LIN {X 0,Y 394.294,Z 695.223,A -85,B 0,C 180,E1 18299.135,E2 18299.135} C_VEL
LIN {X 0,Y 391.517,Z 710.275,A -85,B 0,C 180,E1 18296.546,E2 18296.546} C_VEL
LIN {X 0,Y 389.156,Z 723.905,A -85,B 0,C 180,E1 18293.789,E2 18293.789} C_VEL
LIN {X 0,Y 387.17,Z 736.546,A -85,B 0,C 180,E1 18290.72,E2 18290.72} C_VEL
LIN {X 0,Y 385.749,Z 746.976,A -85,B 0,C 180,E1 18287.654,E2 18287.654} C_VEL
LIN {X 0,Y 384.84,Z 755.495,A -85,B 0,C 180,E1 18284.597,E2 18284.597} C_VEL
LIN {X 0,Y 384.288,Z 762.773,A -85,B 0,C 180,E1 18281.253,E2 18281.253} C_VEL
LIN {X 0,Y 384.081,Z 767.655,A -85,B 0,C 180,E1 18278.232,E2 18278.232} C_VEL
LIN {X 0,Y 384.027,Z 771.125,A -85,B 0,C 180,E1 18275.078,E2 18275.078} C_VEL
LIN {X 0,Y 384.034,Z 772.853,A -85,B 0,C 180,E1 18272.089,E2 18272.089} C_VEL
LIN {X 0,Y 384.041,Z 773.096,A -85,B 0,C 180,E1 18268.956,E2 18268.956} C_VEL
LIN {X 0,Y 384.03,Z 771.796,A -85,B 0,C 180,E1 18265.969,E2 18265.969} C_VEL
LIN {X 0,Y 384.061,Z 768.821,A -85,B 0,C 180,E1 18262.821,E2 18262.821} C_VEL
LIN {X 0,Y 384.195,Z 764.382,A -85,B 0,C 180,E1 18259.807,E2 18259.807} C_VEL
LIN {X 0,Y 384.596,Z 757.969,A -85,B 0,C 180,E1 18256.621,E2 18256.621} C_VEL
LIN {X 0,Y 385.379,Z 749.606,A -85,B 0,C 180,E1 18253.417,E2 18253.417} C_VEL
LIN {X 0,Y 386.587,Z 739.686,A -85,B 0,C 180,E1 18250.352,E2 18250.352} C_VEL
LIN {X 0,Y 388.331,Z 727.636,A -85,B 0,C 180,E1 18247.281,E2 18247.281} C_VEL
LIN {X 0,Y 390.438,Z 714.67,A -85,B 0,C 180,E1 18244.518,E2 18244.518} C_VEL
LIN {X 0,Y 393.123,Z 699.469,A -85,B 0,C 180,E1 18241.766,E2 18241.766} C_VEL
LIN {X 0,Y 396.114,Z 683.012,A -85,B 0,C 180,E1 18239.26,E2 18239.26} C_VEL
LIN {X 0,Y 399.307,Z 665.741,A -85,B 0,C 180,E1 18237.017,E2 18237.017} C_VEL
LIN {X 0,Y 402.758,Z 646.554,A -85,B 0,C 180,E1 18234.921,E2 18234.921} C_VEL
LIN {X 0,Y 406.358,Z 625.751,A -85,B 0,C 180,E1 18233.015,E2 18233.015} C_VEL
LIN {X 0,Y 410.133,Z 603.324,A -85,B 0,C 180,E1 18231.294,E2 18231.294} C_VEL
LIN {X 0,Y 413.644,Z 580.978,A -85,B 0,C 180,E1 18229.895,E2 18229.895} C_VEL
LIN {X 0,Y 417.206,Z 557.129,A -85,B 0,C 180,E1 18228.681,E2 18228.681} C_VEL
LIN {X 0,Y 420.545,Z 532.633,A -85,B 0,C 180,E1 18227.713,E2 18227.713} C_VEL
LIN {X 0,Y 423.355,Z 506.29,A -85,B 0,C 180,E1 18226.922,E2 18226.922} C_VEL
LIN {X 0,Y 425.187,Z 485.655,A -85,B 0,C 180,E1 18226.474,E2 18226.474} C_VEL
LIN {X 0,Y 427.43,Z 463.252,A -85,B 0,C 180,E1 18226.233,E2 18226.233} C_VEL
LIN {X 0,Y 430.001,Z 440.333,A -85,B 0,C 180,E1 18226.045,E2 18226.045} C_VEL
LIN {X 0,Y 437.672,Z 418.91,A -85,B 0,C 180,E1 18225.373,E2 18225.373} C_VEL
LIN {X 0,Y 445.295,Z 397.451,A -85,B 0,C 180,E1 18224.711,E2 18224.711} C_VEL
LIN {X 0,Y 455.695,Z 372.925,A -85,B 0,C 180,E1 18224.152,E2 18224.152} C_VEL
LIN {X 0,Y 470.521,Z 341.939,A -85,B 0,C 180,E1 18223.651,E2 18223.651} C_VEL
LIN {X 0,Y 460.391,Z 331.053,A -85,B 0,C 180,E1 18221.815,E2 18221.815} C_VEL
LIN {X 0,Y 451.953,Z 318.726,A -85,B 0,C 180,E1 18219.908,E2 18219.908} C_VEL
LIN {X 0,Y 445.362,Z 304.779,A -85,B 0,C 180,E1 18217.962,E2 18217.962} C_VEL
LIN {X 0,Y 440.291,Z 291.135,A -85,B 0,C 180,E1 18216.107,E2 18216.107} C_VEL
LIN {X 0,Y 426.278,Z 299.916,A -85,B 0,C 180,E1 18214.584,E2 18214.584} C_VEL
LIN {X 0,Y 421.514,Z 303.016,A -85,B 0,C 180,E1 18214.042,E2 18214.042} C_VEL
LIN {X 0,Y 419.973,Z 303.956,A -85,B 0,C 180,E1 18213.855,E2 18213.855} C_VEL
LIN {X 0,Y 415.952,Z 306.923,A -85,B 0,C 180,E1 18213.399,E2 18213.399} C_VEL
LIN {X 0,Y 413.79,Z 308.018,A -85,B 0,C 180,E1 18213.099,E2 18213.099} C_VEL
LIN {X 0,Y 410.423,Z 310.916,A -85,B 0,C 180,E1 18212.74,E2 18212.74} C_VEL
LIN {X 0,Y 407.643,Z 312.19,A -85,B 0,C 180,E1 18212.324,E2 18212.324} C_VEL
LIN {X 0,Y 407.314,Z 312.632,A -85,B 0,C 180,E1 18212.228,E2 18212.228} C_VEL
LIN {X 0,Y 405.552,Z 347.302,A -85,B 0,C 180,E1 18208.976,E2 18208.976} C_VEL
LIN {X 0,Y 402.812,Z 358.585,A -85,B 0,C 180,E1 18208.28,E2 18208.28} C_VEL
LIN {X 0,Y 397.59,Z 457.682,A -85,B 0,C 180,E1 18205.679,E2 18205.679} C_VEL
LIN {X 0,Y 396.033,Z 507.95,A -85,B 0,C 180,E1 18204.434,E2 18204.434} C_VEL
LIN {X 0,Y 395.904,Z 528.625,A -85,B 0,C 180,E1 18203.798,E2 18203.798} C_VEL
LIN {X 0,Y 395.515,Z 545.902,A -85,B 0,C 180,E1 18202.998,E2 18202.998} C_VEL
LIN {X 0,Y 394.84,Z 562.776,A -85,B 0,C 180,E1 18201.932,E2 18201.932} C_VEL
LIN {X 0,Y 393.999,Z 577.422,A -85,B 0,C 180,E1 18200.732,E2 18200.732} C_VEL
LIN {X 0,Y 392.965,Z 591.658,A -85,B 0,C 180,E1 18199.269,E2 18199.269} C_VEL
LIN {X 0,Y 391.833,Z 604.688,A -85,B 0,C 180,E1 18197.6,E2 18197.6} C_VEL
LIN {X 0,Y 390.654,Z 616.279,A -85,B 0,C 180,E1 18195.741,E2 18195.741} C_VEL
LIN {X 0,Y 389.573,Z 625.958,A -85,B 0,C 180,E1 18193.809,E2 18193.809} C_VEL
LIN {X 0,Y 388.598,Z 634.231,A -85,B 0,C 180,E1 18191.728,E2 18191.728} C_VEL
LIN {X 0,Y 387.758,Z 641.05,A -85,B 0,C 180,E1 18189.498,E2 18189.498} C_VEL
LIN {X 0,Y 387.046,Z 646.284,A -85,B 0,C 180,E1 18187.122,E2 18187.122} C_VEL
LIN {X 0,Y 386.544,Z 649.693,A -85,B 0,C 180,E1 18184.747,E2 18184.747} C_VEL
LIN {X 0,Y 386.218,Z 651.422,A -85,B 0,C 180,E1 18182.373,E2 18182.373} C_VEL
LIN {X 0,Y 386.011,Z 651.4,A -85,B 0,C 180,E1 18179.851,E2 18179.851} C_VEL
LIN {X 0,Y 385.936,Z 649.574,A -85,B 0,C 180,E1 18177.327,E2 18177.327} C_VEL
LIN {X 0,Y 386.012,Z 646.184,A -85,B 0,C 180,E1 18174.947,E2 18174.947} C_VEL
LIN {X 0,Y 386.251,Z 640.868,A -85,B 0,C 180,E1 18172.502,E2 18172.502} C_VEL
LIN {X 0,Y 386.713,Z 633.494,A -85,B 0,C 180,E1 18170.024,E2 18170.024} C_VEL
LIN {X 0,Y 387.328,Z 624.834,A -85,B 0,C 180,E1 18167.779,E2 18167.779} C_VEL
LIN {X 0,Y 388.144,Z 614.206,A -85,B 0,C 180,E1 18165.6,E2 18165.6} C_VEL
LIN {X 0,Y 389.128,Z 602.06,A -85,B 0,C 180,E1 18163.581,E2 18163.581} C_VEL
LIN {X 0,Y 390.161,Z 588.633,A -85,B 0,C 180,E1 18161.781,E2 18161.781} C_VEL
LIN {X 0,Y 391.254,Z 573.412,A -85,B 0,C 180,E1 18160.126,E2 18160.126} C_VEL
LIN {X 0,Y 392.223,Z 557.926,A -85,B 0,C 180,E1 18158.777,E2 18158.777} C_VEL
LIN {X 0,Y 393.053,Z 541.339,A -85,B 0,C 180,E1 18157.647,E2 18157.647} C_VEL
LIN {X 0,Y 393.728,Z 523.341,A -85,B 0,C 180,E1 18156.721,E2 18156.721} C_VEL
LIN {X 0,Y 394.125,Z 505.047,A -85,B 0,C 180,E1 18156.081,E2 18156.081} C_VEL
LIN {X 0,Y 395.755,Z 430.059,A -85,B 0,C 180,E1 18154.443,E2 18154.443} C_VEL
LIN {X 0,Y 396.66,Z 431.556,A -85,B 0,C 180,E1 18154.226,E2 18154.226} C_VEL
LIN {X 0,Y 397.879,Z 431.207,A -85,B 0,C 180,E1 18154.026,E2 18154.026} C_VEL
LIN {X 0,Y 400.105,Z 427.97,A -85,B 0,C 180,E1 18153.765,E2 18153.765} C_VEL
LIN {X 0,Y 403.559,Z 419.262,A -85,B 0,C 180,E1 18153.494,E2 18153.494} C_VEL
LIN {X 0,Y 407.439,Z 406.176,A -85,B 0,C 180,E1 18153.315,E2 18153.315} C_VEL
LIN {X 0,Y 410.429,Z 403.026,A -85,B 0,C 180,E1 18152.938,E2 18152.938} C_VEL
LIN {X 0,Y 413.594,Z 397.112,A -85,B 0,C 180,E1 18152.627,E2 18152.627} C_VEL
LIN {X 0,Y 417.56,Z 386.016,A -85,B 0,C 180,E1 18152.365,E2 18152.365} C_VEL
LIN {X 0,Y 420.1,Z 377.339,A -85,B 0,C 180,E1 18152.251,E2 18152.251} C_VEL
LIN {X 0,Y 423.72,Z 372.276,A -85,B 0,C 180,E1 18151.858,E2 18151.858} C_VEL
LIN {X 0,Y 427.336,Z 364.779,A -85,B 0,C 180,E1 18151.547,E2 18151.547} C_VEL
LIN {X 0,Y 420.508,Z 485.41,A -85,B 0,C 180,E1 18148.882,E2 18148.882} C_VEL
LIN {X 0,Y 419.078,Z 506.712,A -85,B 0,C 180,E1 18148.181,E2 18148.181} C_VEL
LIN {X 0,Y 417.117,Z 526.82,A -85,B 0,C 180,E1 18147.286,E2 18147.286} C_VEL
LIN {X 0,Y 414.553,Z 546.679,A -85,B 0,C 180,E1 18146.141,E2 18146.141} C_VEL
LIN {X 0,Y 411.67,Z 565.181,A -85,B 0,C 180,E1 18144.815,E2 18144.815} C_VEL
LIN {X 0,Y 408.201,Z 584.555,A -85,B 0,C 180,E1 18143.122,E2 18143.122} C_VEL
LIN {X 0,Y 404.781,Z 601.813,A -85,B 0,C 180,E1 18141.312,E2 18141.312} C_VEL
LIN {X 0,Y 401.229,Z 618.426,A -85,B 0,C 180,E1 18139.238,E2 18139.238} C_VEL
LIN {X 0,Y 397.722,Z 634.011,A -85,B 0,C 180,E1 18136.916,E2 18136.916} C_VEL
LIN {X 0,Y 396.207,Z 640.64,A -85,B 0,C 180,E1 18135.799,E2 18135.799} C_VEL
LIN {X 0,Y 394.209,Z 645.664,A -85,B 0,C 180,E1 18134.986,E2 18134.986} C_VEL
LIN {X 0,Y 386.021,Z 658.09,A -85,B 0,C 180,E1 18132.995,E2 18132.995} C_VEL
LIN {X 0,Y 384.095,Z 662.438,A -85,B 0,C 180,E1 18132.085,E2 18132.085} C_VEL
LIN {X 0,Y 381.532,Z 673.871,A -85,B 0,C 180,E1 18129.167,E2 18129.167} C_VEL
LIN {X 0,Y 379.436,Z 684.194,A -85,B 0,C 180,E1 18125.99,E2 18125.99} C_VEL
LIN {X 0,Y 377.914,Z 692.735,A -85,B 0,C 180,E1 18122.717,E2 18122.717} C_VEL
LIN {X 0,Y 376.965,Z 699.299,A -85,B 0,C 180,E1 18119.542,E2 18119.542} C_VEL
LIN {X 0,Y 376.439,Z 704.389,A -85,B 0,C 180,E1 18116.332,E2 18116.332} C_VEL
LIN {X 0,Y 376.179,Z 707.924,A -85,B 0,C 180,E1 18113.124,E2 18113.124} C_VEL
LIN {X 0,Y 376.088,Z 709.954,A -85,B 0,C 180,E1 18109.895,E2 18109.895} C_VEL
LIN {X 0,Y 376.071,Z 710.58,A -85,B 0,C 180,E1 18106.687,E2 18106.687} C_VEL
LIN {X 0,Y 376.1,Z 709.779,A -85,B 0,C 180,E1 18103.687,E2 18103.687} C_VEL
LIN {X 0,Y 376.183,Z 707.48,A -85,B 0,C 180,E1 18100.413,E2 18100.413} C_VEL
LIN {X 0,Y 376.478,Z 703.74,A -85,B 0,C 180,E1 18097.171,E2 18097.171} C_VEL
LIN {X 0,Y 377.042,Z 698.365,A -85,B 0,C 180,E1 18093.954,E2 18093.954} C_VEL
LIN {X 0,Y 378.046,Z 691.428,A -85,B 0,C 180,E1 18090.758,E2 18090.758} C_VEL
LIN {X 0,Y 379.555,Z 682.813,A -85,B 0,C 180,E1 18087.585,E2 18087.585} C_VEL
LIN {X 0,Y 381.686,Z 672.325,A -85,B 0,C 180,E1 18084.438,E2 18084.438} C_VEL
LIN {X 0,Y 384.329,Z 660.268,A -85,B 0,C 180,E1 18081.472,E2 18081.472} C_VEL
LIN {X 0,Y 387.238,Z 647.456,A -85,B 0,C 180,E1 18078.834,E2 18078.834} C_VEL
LIN {X 0,Y 390.705,Z 632.492,A -85,B 0,C 180,E1 18076.232,E2 18076.232} C_VEL
LIN {X 0,Y 394.121,Z 617.507,A -85,B 0,C 180,E1 18074.023,E2 18074.023} C_VEL
LIN {X 0,Y 397.797,Z 600.456,A -85,B 0,C 180,E1 18071.916,E2 18071.916} C_VEL
LIN {X 0,Y 401.228,Z 583.026,A -85,B 0,C 180,E1 18070.114,E2 18070.114} C_VEL
LIN {X 0,Y 404.629,Z 563.988,A -85,B 0,C 180,E1 18068.472,E2 18068.472} C_VEL
LIN {X 0,Y 407.598,Z 544.881,A -85,B 0,C 180,E1 18067.12,E2 18067.12} C_VEL
LIN {X 0,Y 410.182,Z 524.837,A -85,B 0,C 180,E1 18065.979,E2 18065.979} C_VEL
LIN {X 0,Y 412.19,Z 504.088,A -85,B 0,C 180,E1 18065.073,E2 18065.073} C_VEL
LIN {X 0,Y 413.586,Z 483.315,A -85,B 0,C 180,E1 18064.407,E2 18064.407} C_VEL
LIN {X 0,Y 421.708,Z 336.491,A -85,B 0,C 180,E1 18061.21,E2 18061.21} C_VEL
LIN {X 0,Y 425.231,Z 261.966,A -85,B 0,C 180,E1 18059.683,E2 18059.683} C_VEL
LIN {X 0,Y 420.483,Z 255.302,A -85,B 0,C 180,E1 18058.843,E2 18058.843} C_VEL
LIN {X 0,Y 408.107,Z 240.28,A -85,B 0,C 180,E1 18056.6,E2 18056.6} C_VEL
LIN {X 0,Y 394.587,Z 224.674,A -85,B 0,C 180,E1 18053.934,E2 18053.934} C_VEL
LIN {X 0,Y 389.309,Z 215.151,A -85,B 0,C 180,E1 18051.007,E2 18051.007} C_VEL
LIN {X 0,Y 386.424,Z 210.114,A -85,B 0,C 180,E1 18049.3,E2 18049.3} C_VEL
LIN {X 0,Y 384.138,Z 205.838,A -85,B 0,C 180,E1 18047.814,E2 18047.814} C_VEL
LIN {X 0,Y 381.393,Z 201.763,A -85,B 0,C 180,E1 18046.133,E2 18046.133} C_VEL
LIN {X 0,Y 380.79,Z 200.065,A -85,B 0,C 180,E1 18045.579,E2 18045.579} C_VEL
LIN {X 0,Y 378.312,Z 196.942,A -85,B 0,C 180,E1 18044.036,E2 18044.036} C_VEL
LIN {X 0,Y 377.679,Z 194.679,A -85,B 0,C 180,E1 18043.279,E2 18043.279} C_VEL
LIN {X 0,Y 377.659,Z 194.68,A -85,B 0,C 180,E1 18039.254,E2 18039.254} C_VEL
LIN {X 0,Y 377.638,Z 194.679,A -85,B 0,C 180,E1 18035.254,E2 18035.254} C_VEL
LIN {X 0,Y 377.649,Z 194.672,A -85,B 0,C 180,E1 18031.222,E2 18031.222} C_VEL
LIN {X 0,Y 377.68,Z 194.664,A -85,B 0,C 180,E1 18027.258,E2 18027.258} C_VEL
LIN {X 0,Y 377.68,Z 194.664,A -85,B 0,C 180,E1 18023.233,E2 18023.233} C_VEL
LIN {X 0,Y 377.663,Z 194.674,A -85,B 0,C 180,E1 18019.166,E2 18019.166} C_VEL
LIN {X 0,Y 377.64,Z 194.692,A -85,B 0,C 180,E1 18015.196,E2 18015.196} C_VEL
LIN {X 0,Y 377.646,Z 194.695,A -85,B 0,C 180,E1 18011.145,E2 18011.145} C_VEL
LIN {X 0,Y 377.678,Z 194.681,A -85,B 0,C 180,E1 18007.148,E2 18007.148} C_VEL
LIN {X 0,Y 377.679,Z 194.674,A -85,B 0,C 180,E1 18003.036,E2 18003.036} C_VEL
LIN {X 0,Y 377.664,Z 194.674,A -85,B 0,C 180,E1 17998.939,E2 17998.939} C_VEL
LIN {X 0,Y 377.651,Z 194.676,A -85,B 0,C 180,E1 17994.836,E2 17994.836} C_VEL
LIN {X 0,Y 377.696,Z 194.891,A -85,B 0,C 180,E1 17994.532,E2 17994.532} C_VEL
LIN {X 0,Y 378.973,Z 198.234,A -85,B 0,C 180,E1 17993.334,E2 17993.334} C_VEL
LIN {X 0,Y 380.98,Z 200.595,A -85,B 0,C 180,E1 17992.157,E2 17992.157} C_VEL
LIN {X 0,Y 382.561,Z 203.956,A -85,B 0,C 180,E1 17990.978,E2 17990.978} C_VEL
LIN {X 0,Y 384.116,Z 205.937,A -85,B 0,C 180,E1 17990.108,E2 17990.108} C_VEL
LIN {X 0,Y 386.128,Z 209.742,A -85,B 0,C 180,E1 17988.802,E2 17988.802} C_VEL
LIN {X 0,Y 387.146,Z 211.326,A -85,B 0,C 180,E1 17988.228,E2 17988.228} C_VEL
LIN {X 0,Y 390.112,Z 216.657,A -85,B 0,C 180,E1 17986.513,E2 17986.513} C_VEL
LIN {X 0,Y 392.926,Z 221.82,A -85,B 0,C 180,E1 17984.957,E2 17984.957} C_VEL
LIN {X 0,Y 397.5,Z 230.233,A -85,B 0,C 180,E1 17982.583,E2 17982.583} C_VEL
LIN {X 0,Y 403.939,Z 242.972,A -85,B 0,C 180,E1 17979.422,E2 17979.422} C_VEL
LIN {X 0,Y 411.253,Z 258.389,A -85,B 0,C 180,E1 17976.045,E2 17976.045} C_VEL
LIN {X 0,Y 419.116,Z 276.363,A -85,B 0,C 180,E1 17972.586,E2 17972.586} C_VEL
LIN {X 0,Y 421.265,Z 281.573,A -85,B 0,C 180,E1 17971.661,E2 17971.661} C_VEL
LIN {X 0,Y 415.36,Z 329.356,A -85,B 0,C 180,E1 17967.206,E2 17967.206} C_VEL
LIN {X 0,Y 415.071,Z 349.51,A -85,B 0,C 180,E1 17965.103,E2 17965.103} C_VEL
LIN {X 0,Y 416.67,Z 366.69,A -85,B 0,C 180,E1 17963.137,E2 17963.137} C_VEL
LIN {X 0,Y 420.351,Z 383.786,A -85,B 0,C 180,E1 17961.013,E2 17961.013} C_VEL
LIN {X 0,Y 425.59,Z 398.459,A -85,B 0,C 180,E1 17959.045,E2 17959.045} C_VEL
LIN {X 0,Y 432.814,Z 412.394,A -85,B 0,C 180,E1 17957.04,E2 17957.04} C_VEL
LIN {X 0,Y 440.064,Z 422.898,A -85,B 0,C 180,E1 17955.431,E2 17955.431} C_VEL
LIN {X 0,Y 429.597,Z 440.126,A -85,B 0,C 180,E1 17954.798,E2 17954.798} C_VEL
LIN {X 0,Y 424.067,Z 450.967,A -85,B 0,C 180,E1 17954.333,E2 17954.333} C_VEL
LIN {X 0,Y 419.786,Z 478.308,A -85,B 0,C 180,E1 17954.236,E2 17954.236} C_VEL
LIN {X 0,Y 417.756,Z 497.612,A -85,B 0,C 180,E1 17953.966,E2 17953.966} C_VEL
LIN {X 0,Y 415.432,Z 524.064,A -85,B 0,C 180,E1 17953.262,E2 17953.262} C_VEL
LIN {X 0,Y 412.156,Z 549.527,A -85,B 0,C 180,E1 17952.361,E2 17952.361} C_VEL
LIN {X 0,Y 408.586,Z 574.112,A -85,B 0,C 180,E1 17951.215,E2 17951.215} C_VEL
LIN {X 0,Y 405.098,Z 596.15,A -85,B 0,C 180,E1 17949.921,E2 17949.921} C_VEL
LIN {X 0,Y 401.194,Z 619.021,A -85,B 0,C 180,E1 17948.276,E2 17948.276} C_VEL
LIN {X 0,Y 397.38,Z 640.175,A -85,B 0,C 180,E1 17946.427,E2 17946.427} C_VEL
LIN {X 0,Y 393.857,Z 658.978,A -85,B 0,C 180,E1 17944.48,E2 17944.48} C_VEL
LIN {X 0,Y 390.464,Z 676.485,A -85,B 0,C 180,E1 17942.326,E2 17942.326} C_VEL
LIN {X 0,Y 386.973,Z 694.2,A -85,B 0,C 180,E1 17939.741,E2 17939.741} C_VEL
LIN {X 0,Y 383.993,Z 709.585,A -85,B 0,C 180,E1 17937.063,E2 17937.063} C_VEL
LIN {X 0,Y 381.524,Z 723.031,A -85,B 0,C 180,E1 17934.296,E2 17934.296} C_VEL
LIN {X 0,Y 379.365,Z 736.05,A -85,B 0,C 180,E1 17931.093,E2 17931.093} C_VEL
LIN {X 0,Y 377.824,Z 746.727,A -85,B 0,C 180,E1 17927.877,E2 17927.877} C_VEL
LIN {X 0,Y 376.871,Z 755.157,A -85,B 0,C 180,E1 17924.755,E2 17924.755} C_VEL
LIN {X 0,Y 376.319,Z 762.107,A -85,B 0,C 180,E1 17921.494,E2 17921.494} C_VEL
LIN {X 0,Y 376.092,Z 767.2,A -85,B 0,C 180,E1 17918.254,E2 17918.254} C_VEL
LIN {X 0,Y 376.046,Z 770.606,A -85,B 0,C 180,E1 17915.034,E2 17915.034} C_VEL
LIN {X 0,Y 376.056,Z 772.288,A -85,B 0,C 180,E1 17911.828,E2 17911.828} C_VEL
LIN {X 0,Y 376.064,Z 772.416,A -85,B 0,C 180,E1 17908.781,E2 17908.781} C_VEL
LIN {X 0,Y 376.056,Z 771.015,A -85,B 0,C 180,E1 17905.73,E2 17905.73} C_VEL
LIN {X 0,Y 376.077,Z 767.954,A -85,B 0,C 180,E1 17902.514,E2 17902.514} C_VEL
LIN {X 0,Y 376.254,Z 763.134,A -85,B 0,C 180,E1 17899.279,E2 17899.279} C_VEL
LIN {X 0,Y 376.709,Z 756.527,A -85,B 0,C 180,E1 17896.023,E2 17896.023} C_VEL
LIN {X 0,Y 377.59,Z 747.944,A -85,B 0,C 180,E1 17892.748,E2 17892.748} C_VEL
LIN {X 0,Y 378.938,Z 737.8,A -85,B 0,C 180,E1 17889.617,E2 17889.617} C_VEL
LIN {X 0,Y 380.869,Z 725.502,A -85,B 0,C 180,E1 17886.482,E2 17886.482} C_VEL
LIN {X 0,Y 383.337,Z 711.485,A -85,B 0,C 180,E1 17883.511,E2 17883.511} C_VEL
LIN {X 0,Y 386.118,Z 696.75,A -85,B 0,C 180,E1 17880.867,E2 17880.867} C_VEL
LIN {X 0,Y 389.365,Z 680.005,A -85,B 0,C 180,E1 17878.324,E2 17878.324} C_VEL
LIN {X 0,Y 392.833,Z 662.18,A -85,B 0,C 180,E1 17876.035,E2 17876.035} C_VEL
LIN {X 0,Y 396.388,Z 643.433,A -85,B 0,C 180,E1 17874.004,E2 17874.004} C_VEL
LIN {X 0,Y 400.236,Z 622.112,A -85,B 0,C 180,E1 17872.08,E2 17872.08} C_VEL
LIN {X 0,Y 404.134,Z 599.984,A -85,B 0,C 180,E1 17870.4,E2 17870.4} C_VEL
LIN {X 0,Y 407.82,Z 577.642,A -85,B 0,C 180,E1 17869.017,E2 17869.017} C_VEL
LIN {X 0,Y 411.567,Z 553.285,A -85,B 0,C 180,E1 17867.799,E2 17867.799} C_VEL
LIN {X 0,Y 415.188,Z 527.849,A -85,B 0,C 180,E1 17866.818,E2 17866.818} C_VEL
LIN {X 0,Y 418.115,Z 500.137,A -85,B 0,C 180,E1 17866.003,E2 17866.003} C_VEL
LIN {X 0,Y 420.284,Z 477.679,A -85,B 0,C 180,E1 17865.589,E2 17865.589} C_VEL
LIN {X 0,Y 424.677,Z 438.091,A -85,B 0,C 180,E1 17865.268,E2 17865.268} C_VEL
LIN {X 0,Y 431.691,Z 418.214,A -85,B 0,C 180,E1 17864.679,E2 17864.679} C_VEL
LIN {X 0,Y 439.368,Z 396.741,A -85,B 0,C 180,E1 17864.018,E2 17864.018} C_VEL
LIN {X 0,Y 449.791,Z 372.162,A -85,B 0,C 180,E1 17863.465,E2 17863.465} C_VEL
LIN {X 0,Y 462.548,Z 345.265,A -85,B 0,C 180,E1 17863.027,E2 17863.027} C_VEL
LIN {X 0,Y 452.399,Z 333.261,A -85,B 0,C 180,E1 17861.026,E2 17861.026} C_VEL
LIN {X 0,Y 445.331,Z 321.899,A -85,B 0,C 180,E1 17859.282,E2 17859.282} C_VEL
LIN {X 0,Y 438.364,Z 305.771,A -85,B 0,C 180,E1 17857.024,E2 17857.024} C_VEL
LIN {X 0,Y 436.404,Z 300.371,A -85,B 0,C 180,E1 17856.276,E2 17856.276} C_VEL
LIN {X 0,Y 425.723,Z 307.062,A -85,B 0,C 180,E1 17855.128,E2 17855.128} C_VEL
LIN {X 0,Y 420.158,Z 310.571,A -85,B 0,C 180,E1 17854.497,E2 17854.497} C_VEL
LIN {X 0,Y 415.363,Z 313.838,A -85,B 0,C 180,E1 17853.949,E2 17853.949} C_VEL
LIN {X 0,Y 413.598,Z 314.99,A -85,B 0,C 180,E1 17853.735,E2 17853.735} C_VEL
LIN {X 0,Y 409.032,Z 318.296,A -85,B 0,C 180,E1 17853.199,E2 17853.199} C_VEL
LIN {X 0,Y 407.617,Z 318.959,A -85,B 0,C 180,E1 17852.994,E2 17852.994} C_VEL
LIN {X 0,Y 403.474,Z 322.407,A -85,B 0,C 180,E1 17852.53,E2 17852.53} C_VEL
LIN {X 0,Y 400.99,Z 323.574,A -85,B 0,C 180,E1 17852.122,E2 17852.122} C_VEL
LIN {X 0,Y 399.312,Z 349.803,A -85,B 0,C 180,E1 17849.638,E2 17849.638} C_VEL
LIN {X 0,Y 396.522,Z 361.178,A -85,B 0,C 180,E1 17848.951,E2 17848.951} C_VEL
LIN {X 0,Y 390.925,Z 456.49,A -85,B 0,C 180,E1 17846.343,E2 17846.343} C_VEL
LIN {X 0,Y 389.035,Z 507.853,A -85,B 0,C 180,E1 17845.01,E2 17845.01} C_VEL
LIN {X 0,Y 388.84,Z 529.87,A -85,B 0,C 180,E1 17844.319,E2 17844.319} C_VEL
LIN {X 0,Y 388.427,Z 547.028,A -85,B 0,C 180,E1 17843.514,E2 17843.514} C_VEL
LIN {X 0,Y 387.687,Z 563.772,A -85,B 0,C 180,E1 17842.438,E2 17842.438} C_VEL
LIN {X 0,Y 386.806,Z 578.646,A -85,B 0,C 180,E1 17841.216,E2 17841.216} C_VEL
LIN {X 0,Y 385.732,Z 592.364,A -85,B 0,C 180,E1 17839.79,E2 17839.79} C_VEL
LIN {X 0,Y 384.469,Z 606.004,A -85,B 0,C 180,E1 17838.027,E2 17838.027} C_VEL
LIN {X 0,Y 383.256,Z 617.265,A -85,B 0,C 180,E1 17836.209,E2 17836.209} C_VEL
LIN {X 0,Y 382.077,Z 627.029,A -85,B 0,C 180,E1 17834.24,E2 17834.24} C_VEL
LIN {X 0,Y 381.016,Z 635.418,A -85,B 0,C 180,E1 17832.118,E2 17832.118} C_VEL
LIN {X 0,Y 380.096,Z 642.326,A -85,B 0,C 180,E1 17829.845,E2 17829.845} C_VEL
LIN {X 0,Y 379.306,Z 647.611,A -85,B 0,C 180,E1 17827.421,E2 17827.421} C_VEL
LIN {X 0,Y 378.746,Z 651.072,A -85,B 0,C 180,E1 17824.997,E2 17824.997} C_VEL
LIN {X 0,Y 378.376,Z 652.823,A -85,B 0,C 180,E1 17822.574,E2 17822.574} C_VEL
LIN {X 0,Y 378.153,Z 652.892,A -85,B 0,C 180,E1 17820.151,E2 17820.151} C_VEL
LIN {X 0,Y 378.046,Z 651.158,A -85,B 0,C 180,E1 17817.574,E2 17817.574} C_VEL
LIN {X 0,Y 378.114,Z 647.611,A -85,B 0,C 180,E1 17814.993,E2 17814.993} C_VEL
LIN {X 0,Y 378.347,Z 642.455,A -85,B 0,C 180,E1 17812.559,E2 17812.559} C_VEL
LIN {X 0,Y 378.792,Z 635.397,A -85,B 0,C 180,E1 17810.12,E2 17810.12} C_VEL
LIN {X 0,Y 379.411,Z 626.846,A -85,B 0,C 180,E1 17807.829,E2 17807.829} C_VEL
LIN {X 0,Y 380.208,Z 616.802,A -85,B 0,C 180,E1 17805.688,E2 17805.688} C_VEL
LIN {X 0,Y 381.239,Z 604.343,A -85,B 0,C 180,E1 17803.545,E2 17803.545} C_VEL
LIN {X 0,Y 382.319,Z 590.976,A -85,B 0,C 180,E1 17801.685,E2 17801.685} C_VEL
LIN {X 0,Y 383.417,Z 576.209,A -85,B 0,C 180,E1 17800.024,E2 17800.024} C_VEL
LIN {X 0,Y 384.455,Z 560.536,A -85,B 0,C 180,E1 17798.601,E2 17798.601} C_VEL
LIN {X 0,Y 385.347,Z 543.835,A -85,B 0,C 180,E1 17797.417,E2 17797.417} C_VEL
LIN {X 0,Y 386.073,Z 525.483,A -85,B 0,C 180,E1 17796.436,E2 17796.436} C_VEL
LIN {X 0,Y 386.515,Z 507.417,A -85,B 0,C 180,E1 17795.768,E2 17795.768} C_VEL
LIN {X 0,Y 387.449,Z 460.917,A -85,B 0,C 180,E1 17794.695,E2 17794.695} C_VEL
LIN {X 0,Y 388.413,Z 462.419,A -85,B 0,C 180,E1 17794.457,E2 17794.457} C_VEL
LIN {X 0,Y 389.885,Z 461.841,A -85,B 0,C 180,E1 17794.22,E2 17794.22} C_VEL
LIN {X 0,Y 392.195,Z 458.299,A -85,B 0,C 180,E1 17793.961,E2 17793.961} C_VEL
LIN {X 0,Y 395.8,Z 449.132,A -85,B 0,C 180,E1 17793.699,E2 17793.699} C_VEL
LIN {X 0,Y 399.044,Z 438.423,A -85,B 0,C 180,E1 17793.552,E2 17793.552} C_VEL
LIN {X 0,Y 401.952,Z 435.45,A -85,B 0,C 180,E1 17793.175,E2 17793.175} C_VEL
LIN {X 0,Y 405.127,Z 429.765,A -85,B 0,C 180,E1 17792.862,E2 17792.862} C_VEL
LIN {X 0,Y 409.11,Z 419.049,A -85,B 0,C 180,E1 17792.6,E2 17792.6} C_VEL
LIN {X 0,Y 411.545,Z 410.947,A -85,B 0,C 180,E1 17792.489,E2 17792.489} C_VEL
LIN {X 0,Y 415.328,Z 405.813,A -85,B 0,C 180,E1 17792.07,E2 17792.07} C_VEL
LIN {X 0,Y 419.194,Z 397.702,A -85,B 0,C 180,E1 17791.75,E2 17791.75} C_VEL
LIN {X 0,Y 420.085,Z 395.468,A -85,B 0,C 180,E1 17791.686,E2 17791.686} C_VEL
LIN {X 0,Y 414.518,Z 487.506,A -85,B 0,C 180,E1 17789.574,E2 17789.574} C_VEL
LIN {X 0,Y 413.014,Z 508.69,A -85,B 0,C 180,E1 17788.861,E2 17788.861} C_VEL
LIN {X 0,Y 410.908,Z 528.915,A -85,B 0,C 180,E1 17787.936,E2 17787.936} C_VEL
LIN {X 0,Y 408.213,Z 548.691,A -85,B 0,C 180,E1 17786.768,E2 17786.768} C_VEL
LIN {X 0,Y 405.061,Z 567.769,A -85,B 0,C 180,E1 17785.364,E2 17785.364} C_VEL
LIN {X 0,Y 401.673,Z 585.771,A -85,B 0,C 180,E1 17783.757,E2 17783.757} C_VEL
LIN {X 0,Y 397.947,Z 603.527,A -85,B 0,C 180,E1 17781.853,E2 17781.853} C_VEL
LIN {X 0,Y 394.137,Z 620.418,A -85,B 0,C 180,E1 17779.692,E2 17779.692} C_VEL
LIN {X 0,Y 390.361,Z 636.323,A -85,B 0,C 180,E1 17777.252,E2 17777.252} C_VEL
LIN {X 0,Y 386.927,Z 650.497,A -85,B 0,C 180,E1 17774.659,E2 17774.659} C_VEL
LIN {X 0,Y 384.095,Z 662.438,A -85,B 0,C 180,E1 17772.085,E2 17772.085} C_VEL
LIN {X 0,Y 382.219,Z 666.725,A -85,B 0,C 180,E1 17771.151,E2 17771.151} C_VEL
LIN {X 0,Y 374.044,Z 677.649,A -85,B 0,C 180,E1 17768.689,E2 17768.689} C_VEL
LIN {X 0,Y 372.662,Z 680.655,A -85,B 0,C 180,E1 17767.802,E2 17767.802} C_VEL
LIN {X 0,Y 370.754,Z 690.001,A -85,B 0,C 180,E1 17764.495,E2 17764.495} C_VEL
LIN {X 0,Y 369.451,Z 697.537,A -85,B 0,C 180,E1 17761.126,E2 17761.126} C_VEL
LIN {X 0,Y 368.691,Z 703.257,A -85,B 0,C 180,E1 17757.804,E2 17757.804} C_VEL
LIN {X 0,Y 368.317,Z 707.379,A -85,B 0,C 180,E1 17754.541,E2 17754.541} C_VEL
LIN {X 0,Y 368.15,Z 709.971,A -85,B 0,C 180,E1 17751.32,E2 17751.32} C_VEL
LIN {X 0,Y 368.1,Z 711.135,A -85,B 0,C 180,E1 17748.039,E2 17748.039} C_VEL
LIN {X 0,Y 368.111,Z 710.908,A -85,B 0,C 180,E1 17744.766,E2 17744.766} C_VEL
LIN {X 0,Y 368.176,Z 709.219,A -85,B 0,C 180,E1 17741.594,E2 17741.594} C_VEL
LIN {X 0,Y 368.383,Z 706.003,A -85,B 0,C 180,E1 17738.271,E2 17738.271} C_VEL
LIN {X 0,Y 368.887,Z 701.327,A -85,B 0,C 180,E1 17734.976,E2 17734.976} C_VEL
LIN {X 0,Y 369.758,Z 694.991,A -85,B 0,C 180,E1 17731.705,E2 17731.705} C_VEL
LIN {X 0,Y 371.144,Z 686.999,A -85,B 0,C 180,E1 17728.457,E2 17728.457} C_VEL
LIN {X 0,Y 373.158,Z 677.222,A -85,B 0,C 180,E1 17725.236,E2 17725.236} C_VEL
LIN {X 0,Y 375.569,Z 666.667,A -85,B 0,C 180,E1 17722.351,E2 17722.351} C_VEL
LIN {X 0,Y 378.728,Z 653.396,A -85,B 0,C 180,E1 17719.351,E2 17719.351} C_VEL
LIN {X 0,Y 381.919,Z 640.107,A -85,B 0,C 180,E1 17716.835,E2 17716.835} C_VEL
LIN {X 0,Y 385.629,Z 624.628,A -85,B 0,C 180,E1 17714.357,E2 17714.357} C_VEL
LIN {X 0,Y 389.298,Z 608.721,A -85,B 0,C 180,E1 17712.204,E2 17712.204} C_VEL
LIN {X 0,Y 393.076,Z 591.329,A -85,B 0,C 180,E1 17710.226,E2 17710.226} C_VEL
LIN {X 0,Y 396.501,Z 573.566,A -85,B 0,C 180,E1 17708.553,E2 17708.553} C_VEL
LIN {X 0,Y 399.657,Z 555.156,A -85,B 0,C 180,E1 17707.106,E2 17707.106} C_VEL
LIN {X 0,Y 402.453,Z 536.163,A -85,B 0,C 180,E1 17705.878,E2 17705.878} C_VEL
LIN {X 0,Y 404.909,Z 515.539,A -85,B 0,C 180,E1 17704.828,E2 17704.828} C_VEL
LIN {X 0,Y 406.676,Z 495.118,A -85,B 0,C 180,E1 17704.047,E2 17704.047} C_VEL
LIN {X 0,Y 408.164,Z 468.968,A -85,B 0,C 180,E1 17703.347,E2 17703.347} C_VEL
LIN {X 0,Y 416.618,Z 324.474,A -85,B 0,C 180,E1 17700.193,E2 17700.193} C_VEL
LIN {X 0,Y 419.477,Z 265.617,A -85,B 0,C 180,E1 17698.971,E2 17698.971} C_VEL
LIN {X 0,Y 409.618,Z 252.975,A -85,B 0,C 180,E1 17697.179,E2 17697.179} C_VEL
LIN {X 0,Y 395.94,Z 236.904,A -85,B 0,C 180,E1 17694.529,E2 17694.529} C_VEL
LIN {X 0,Y 388.107,Z 228.075,A -85,B 0,C 180,E1 17692.878,E2 17692.878} C_VEL
LIN {X 0,Y 384.534,Z 221.418,A -85,B 0,C 180,E1 17690.793,E2 17690.793} C_VEL
LIN {X 0,Y 381.549,Z 216.236,A -85,B 0,C 180,E1 17689.001,E2 17689.001} C_VEL
LIN {X 0,Y 378.978,Z 211.546,A -85,B 0,C 180,E1 17687.309,E2 17687.309} C_VEL
LIN {X 0,Y 376.66,Z 207.794,A -85,B 0,C 180,E1 17685.786,E2 17685.786} C_VEL
LIN {X 0,Y 375.966,Z 206.356,A -85,B 0,C 180,E1 17685.241,E2 17685.241} C_VEL
LIN {X 0,Y 373.636,Z 202.992,A -85,B 0,C 180,E1 17683.664,E2 17683.664} C_VEL
LIN {X 0,Y 372.873,Z 201.079,A -85,B 0,C 180,E1 17682.931,E2 17682.931} C_VEL
LIN {X 0,Y 370.344,Z 197.878,A -85,B 0,C 180,E1 17681.128,E2 17681.128} C_VEL
LIN {X 0,Y 369.75,Z 195.652,A -85,B 0,C 180,E1 17680.263,E2 17680.263} C_VEL
LIN {X 0,Y 369.721,Z 195.655,A -85,B 0,C 180,E1 17676.303,E2 17676.303} C_VEL
LIN {X 0,Y 369.699,Z 195.657,A -85,B 0,C 180,E1 17672.166,E2 17672.166} C_VEL
LIN {X 0,Y 369.722,Z 195.658,A -85,B 0,C 180,E1 17668.162,E2 17668.162} C_VEL
LIN {X 0,Y 369.739,Z 195.663,A -85,B 0,C 180,E1 17664.101,E2 17664.101} C_VEL
LIN {X 0,Y 369.747,Z 195.677,A -85,B 0,C 180,E1 17660.087,E2 17660.087} C_VEL
LIN {X 0,Y 369.718,Z 195.681,A -85,B 0,C 180,E1 17656.013,E2 17656.013} C_VEL
LIN {X 0,Y 369.696,Z 195.668,A -85,B 0,C 180,E1 17652.02,E2 17652.02} C_VEL
LIN {X 0,Y 369.714,Z 195.659,A -85,B 0,C 180,E1 17647.928,E2 17647.928} C_VEL
LIN {X 0,Y 369.735,Z 195.654,A -85,B 0,C 180,E1 17643.877,E2 17643.877} C_VEL
LIN {X 0,Y 369.747,Z 195.653,A -85,B 0,C 180,E1 17639.846,E2 17639.846} C_VEL
LIN {X 0,Y 369.739,Z 195.824,A -85,B 0,C 180,E1 17637.521,E2 17637.521} C_VEL
LIN {X 0,Y 371.037,Z 199.144,A -85,B 0,C 180,E1 17636.138,E2 17636.138} C_VEL
LIN {X 0,Y 373.135,Z 201.376,A -85,B 0,C 180,E1 17634.773,E2 17634.773} C_VEL
LIN {X 0,Y 374.644,Z 204.97,A -85,B 0,C 180,E1 17633.411,E2 17633.411} C_VEL
LIN {X 0,Y 376.357,Z 207.084,A -85,B 0,C 180,E1 17632.367,E2 17632.367} C_VEL
LIN {X 0,Y 378.221,Z 210.707,A -85,B 0,C 180,E1 17631.027,E2 17631.027} C_VEL
LIN {X 0,Y 379.464,Z 212.448,A -85,B 0,C 180,E1 17630.292,E2 17630.292} C_VEL
LIN {X 0,Y 381.782,Z 216.509,A -85,B 0,C 180,E1 17628.826,E2 17628.826} C_VEL
LIN {X 0,Y 385.394,Z 223.175,A -85,B 0,C 180,E1 17626.65,E2 17626.65} C_VEL
LIN {X 0,Y 388.198,Z 228.356,A -85,B 0,C 180,E1 17625.075,E2 17625.075} C_VEL
LIN {X 0,Y 392.459,Z 236.271,A -85,B 0,C 180,E1 17622.811,E2 17622.811} C_VEL
LIN {X 0,Y 398.821,Z 249.054,A -85,B 0,C 180,E1 17619.606,E2 17619.606} C_VEL
LIN {X 0,Y 405.76,Z 263.875,A -85,B 0,C 180,E1 17616.319,E2 17616.319} C_VEL
LIN {X 0,Y 413.337,Z 281.418,A -85,B 0,C 180,E1 17612.897,E2 17612.897} C_VEL
LIN {X 0,Y 414.975,Z 285.745,A -85,B 0,C 180,E1 17612.133,E2 17612.133} C_VEL
LIN {X 0,Y 409.009,Z 331.724,A -85,B 0,C 180,E1 17607.797,E2 17607.797} C_VEL
LIN {X 0,Y 408.555,Z 351.965,A -85,B 0,C 180,E1 17605.66,E2 17605.66} C_VEL
LIN {X 0,Y 410.094,Z 370.019,A -85,B 0,C 180,E1 17603.57,E2 17603.57} C_VEL
LIN {X 0,Y 413.802,Z 387.726,A -85,B 0,C 180,E1 17601.338,E2 17601.338} C_VEL
LIN {X 0,Y 419.354,Z 403.358,A -85,B 0,C 180,E1 17599.21,E2 17599.21} C_VEL
LIN {X 0,Y 427.057,Z 418.072,A -85,B 0,C 180,E1 17597.054,E2 17597.054} C_VEL
LIN {X 0,Y 431.696,Z 425.014,A -85,B 0,C 180,E1 17595.986,E2 17595.986} C_VEL
LIN {X 0,Y 421.313,Z 442.703,A -85,B 0,C 180,E1 17595.298,E2 17595.298} C_VEL
LIN {X 0,Y 418.559,Z 448.366,A -85,B 0,C 180,E1 17595.068,E2 17595.068} C_VEL
LIN {X 0,Y 414.001,Z 476.945,A -85,B 0,C 180,E1 17594.984,E2 17594.984} C_VEL
LIN {X 0,Y 411.728,Z 497.471,A -85,B 0,C 180,E1 17594.695,E2 17594.695} C_VEL
LIN {X 0,Y 409.224,Z 523.884,A -85,B 0,C 180,E1 17593.967,E2 17593.967} C_VEL
LIN {X 0,Y 405.667,Z 550.336,A -85,B 0,C 180,E1 17593.009,E2 17593.009} C_VEL
LIN {X 0,Y 401.994,Z 574.532,A -85,B 0,C 180,E1 17591.854,E2 17591.854} C_VEL
LIN {X 0,Y 398.132,Z 597.699,A -85,B 0,C 180,E1 17590.453,E2 17590.453} C_VEL
LIN {X 0,Y 394.138,Z 620.044,A -85,B 0,C 180,E1 17588.799,E2 17588.799} C_VEL
LIN {X 0,Y 390.185,Z 641.11,A -85,B 0,C 180,E1 17586.917,E2 17586.917} C_VEL
LIN {X 0,Y 386.428,Z 660.306,A -85,B 0,C 180,E1 17584.877,E2 17584.877} C_VEL
LIN {X 0,Y 382.486,Z 679.662,A -85,B 0,C 180,E1 17582.398,E2 17582.398} C_VEL
LIN {X 0,Y 379.108,Z 695.976,A -85,B 0,C 180,E1 17579.899,E2 17579.899} C_VEL
LIN {X 0,Y 376.099,Z 710.869,A -85,B 0,C 180,E1 17577.21,E2 17577.21} C_VEL
LIN {X 0,Y 373.405,Z 724.914,A -85,B 0,C 180,E1 17574.185,E2 17574.185} C_VEL
LIN {X 0,Y 371.467,Z 736.098,A -85,B 0,C 180,E1 17571.307,E2 17571.307} C_VEL
LIN {X 0,Y 369.905,Z 746.462,A -85,B 0,C 180,E1 17568.11,E2 17568.11} C_VEL
LIN {X 0,Y 368.904,Z 754.826,A -85,B 0,C 180,E1 17564.921,E2 17564.921} C_VEL
LIN {X 0,Y 368.333,Z 761.72,A -85,B 0,C 180,E1 17561.588,E2 17561.588} C_VEL
LIN {X 0,Y 368.104,Z 766.737,A -85,B 0,C 180,E1 17558.277,E2 17558.277} C_VEL
LIN {X 0,Y 368.066,Z 769.949,A -85,B 0,C 180,E1 17555.143,E2 17555.143} C_VEL
LIN {X 0,Y 368.083,Z 771.633,A -85,B 0,C 180,E1 17551.868,E2 17551.868} C_VEL
LIN {X 0,Y 368.09,Z 771.756,A -85,B 0,C 180,E1 17548.755,E2 17548.755} C_VEL
LIN {X 0,Y 368.078,Z 770.349,A -85,B 0,C 180,E1 17545.638,E2 17545.638} C_VEL
LIN {X 0,Y 368.095,Z 767.267,A -85,B 0,C 180,E1 17542.351,E2 17542.351} C_VEL
LIN {X 0,Y 368.265,Z 762.701,A -85,B 0,C 180,E1 17539.202,E2 17539.202} C_VEL
LIN {X 0,Y 368.736,Z 756.164,A -85,B 0,C 180,E1 17535.874,E2 17535.874} C_VEL
LIN {X 0,Y 369.601,Z 748.105,A -85,B 0,C 180,E1 17532.688,E2 17532.688} C_VEL
LIN {X 0,Y 370.99,Z 738.165,A -85,B 0,C 180,E1 17529.49,E2 17529.49} C_VEL
LIN {X 0,Y 372.988,Z 726.042,A -85,B 0,C 180,E1 17526.29,E2 17526.29} C_VEL
LIN {X 0,Y 375.405,Z 713.1,A -85,B 0,C 180,E1 17523.419,E2 17523.419} C_VEL
LIN {X 0,Y 378.444,Z 697.8,A -85,B 0,C 180,E1 17520.566,E2 17520.566} C_VEL
LIN {X 0,Y 381.825,Z 681.38,A -85,B 0,C 180,E1 17517.976,E2 17517.976} C_VEL
LIN {X 0,Y 385.556,Z 663.286,A -85,B 0,C 180,E1 17515.574,E2 17515.574} C_VEL
LIN {X 0,Y 389.406,Z 644.094,A -85,B 0,C 180,E1 17513.437,E2 17513.437} C_VEL
LIN {X 0,Y 393.592,Z 622.22,A -85,B 0,C 180,E1 17511.416,E2 17511.416} C_VEL
LIN {X 0,Y 397.788,Z 599.364,A -85,B 0,C 180,E1 17509.666,E2 17509.666} C_VEL
LIN {X 0,Y 401.898,Z 575.602,A -85,B 0,C 180,E1 17508.184,E2 17508.184} C_VEL
LIN {X 0,Y 405.965,Z 550.427,A -85,B 0,C 180,E1 17506.933,E2 17506.933} C_VEL
LIN {X 0,Y 409.76,Z 524.453,A -85,B 0,C 180,E1 17505.946,E2 17505.946} C_VEL
LIN {X 0,Y 412.776,Z 496.488,A -85,B 0,C 180,E1 17505.13,E2 17505.13} C_VEL
LIN {X 0,Y 415.37,Z 472.026,A -85,B 0,C 180,E1 17504.725,E2 17504.725} C_VEL
LIN {X 0,Y 419.523,Z 436.035,A -85,B 0,C 180,E1 17504.461,E2 17504.461} C_VEL
LIN {X 0,Y 420.093,Z 433.059,A -85,B 0,C 180,E1 17504.436,E2 17504.436} C_VEL
LIN {X 0,Y 425.772,Z 417.581,A -85,B 0,C 180,E1 17503.964,E2 17503.964} C_VEL
LIN {X 0,Y 433.499,Z 396.102,A -85,B 0,C 180,E1 17503.306,E2 17503.306} C_VEL
LIN {X 0,Y 443.936,Z 371.525,A -85,B 0,C 180,E1 17502.757,E2 17502.757} C_VEL
LIN {X 0,Y 454.722,Z 348.413,A -85,B 0,C 180,E1 17502.372,E2 17502.372} C_VEL
LIN {X 0,Y 445.077,Z 336.031,A -85,B 0,C 180,E1 17500.314,E2 17500.314} C_VEL
LIN {X 0,Y 437.988,Z 323.313,A -85,B 0,C 180,E1 17498.384,E2 17498.384} C_VEL
LIN {X 0,Y 432.505,Z 309.495,A -85,B 0,C 180,E1 17496.437,E2 17496.437} C_VEL
LIN {X 0,Y 419.582,Z 317.755,A -85,B 0,C 180,E1 17495.05,E2 17495.05} C_VEL
LIN {X 0,Y 413.98,Z 321.402,A -85,B 0,C 180,E1 17494.413,E2 17494.413} C_VEL
LIN {X 0,Y 409.175,Z 324.79,A -85,B 0,C 180,E1 17493.858,E2 17493.858} C_VEL
LIN {X 0,Y 407.669,Z 325.668,A -85,B 0,C 180,E1 17493.662,E2 17493.662} C_VEL
LIN {X 0,Y 403.571,Z 328.881,A -85,B 0,C 180,E1 17493.198,E2 17493.198} C_VEL
LIN {X 0,Y 401.138,Z 330.242,A -85,B 0,C 180,E1 17492.86,E2 17492.86} C_VEL
LIN {X 0,Y 397.244,Z 333.52,A -85,B 0,C 180,E1 17492.419,E2 17492.419} C_VEL
LIN {X 0,Y 394.709,Z 334.701,A -85,B 0,C 180,E1 17492.009,E2 17492.009} C_VEL
LIN {X 0,Y 393.412,Z 351.736,A -85,B 0,C 180,E1 17490.381,E2 17490.381} C_VEL
LIN {X 0,Y 390.414,Z 363.495,A -85,B 0,C 180,E1 17489.669,E2 17489.669} C_VEL
LIN {X 0,Y 384.226,Z 458.709,A -85,B 0,C 180,E1 17486.959,E2 17486.959} C_VEL
LIN {X 0,Y 382.108,Z 509.638,A -85,B 0,C 180,E1 17485.57,E2 17485.57} C_VEL
LIN {X 0,Y 381.872,Z 531.291,A -85,B 0,C 180,E1 17484.87,E2 17484.87} C_VEL
LIN {X 0,Y 381.413,Z 548.289,A -85,B 0,C 180,E1 17484.056,E2 17484.056} C_VEL
LIN {X 0,Y 380.557,Z 566.137,A -85,B 0,C 180,E1 17482.882,E2 17482.882} C_VEL
LIN {X 0,Y 379.596,Z 580.785,A -85,B 0,C 180,E1 17481.639,E2 17481.639} C_VEL
LIN {X 0,Y 378.311,Z 595.835,A -85,B 0,C 180,E1 17480.014,E2 17480.014} C_VEL
LIN {X 0,Y 377.039,Z 608.524,A -85,B 0,C 180,E1 17478.309,E2 17478.309} C_VEL
LIN {X 0,Y 375.684,Z 619.931,A -85,B 0,C 180,E1 17476.386,E2 17476.386} C_VEL
LIN {X 0,Y 374.445,Z 629.527,A -85,B 0,C 180,E1 17474.378,E2 17474.378} C_VEL
LIN {X 0,Y 373.315,Z 637.705,A -85,B 0,C 180,E1 17472.215,E2 17472.215} C_VEL
LIN {X 0,Y 372.327,Z 644.386,A -85,B 0,C 180,E1 17469.896,E2 17469.896} C_VEL
LIN {X 0,Y 371.493,Z 649.507,A -85,B 0,C 180,E1 17467.422,E2 17467.422} C_VEL
LIN {X 0,Y 370.897,Z 652.787,A -85,B 0,C 180,E1 17464.948,E2 17464.948} C_VEL
LIN {X 0,Y 370.499,Z 654.344,A -85,B 0,C 180,E1 17462.474,E2 17462.474} C_VEL
LIN {X 0,Y 370.26,Z 654.207,A -85,B 0,C 180,E1 17459.999,E2 17459.999} C_VEL
LIN {X 0,Y 370.154,Z 652.283,A -85,B 0,C 180,E1 17457.368,E2 17457.368} C_VEL
LIN {X 0,Y 370.224,Z 648.78,A -85,B 0,C 180,E1 17454.886,E2 17454.886} C_VEL
LIN {X 0,Y 370.468,Z 643.479,A -85,B 0,C 180,E1 17452.4,E2 17452.4} C_VEL
LIN {X 0,Y 370.94,Z 636.279,A -85,B 0,C 180,E1 17449.909,E2 17449.909} C_VEL
LIN {X 0,Y 371.596,Z 627.576,A -85,B 0,C 180,E1 17447.569,E2 17447.569} C_VEL
LIN {X 0,Y 372.435,Z 617.324,A -85,B 0,C 180,E1 17445.382,E2 17445.382} C_VEL
LIN {X 0,Y 373.479,Z 605.139,A -85,B 0,C 180,E1 17443.274,E2 17443.274} C_VEL
LIN {X 0,Y 374.541,Z 592.43,A -85,B 0,C 180,E1 17441.477,E2 17441.477} C_VEL
LIN {X 0,Y 375.694,Z 577.424,A -85,B 0,C 180,E1 17439.758,E2 17439.758} C_VEL
LIN {X 0,Y 376.798,Z 561.324,A -85,B 0,C 180,E1 17438.273,E2 17438.273} C_VEL
LIN {X 0,Y 377.7,Z 544.998,A -85,B 0,C 180,E1 17437.098,E2 17437.098} C_VEL
LIN {X 0,Y 378.457,Z 526.595,A -85,B 0,C 180,E1 17436.095,E2 17436.095} C_VEL
LIN {X 0,Y 378.917,Z 508.579,A -85,B 0,C 180,E1 17435.415,E2 17435.415} C_VEL
LIN {X 0,Y 379.145,Z 490.194,A -85,B 0,C 180,E1 17434.959,E2 17434.959} C_VEL
LIN {X 0,Y 380.144,Z 492.003,A -85,B 0,C 180,E1 17434.696,E2 17434.696} C_VEL
LIN {X 0,Y 381.531,Z 491.652,A -85,B 0,C 180,E1 17434.462,E2 17434.462} C_VEL
LIN {X 0,Y 383.712,Z 488.59,A -85,B 0,C 180,E1 17434.204,E2 17434.204} C_VEL
LIN {X 0,Y 387.24,Z 480.148,A -85,B 0,C 180,E1 17433.937,E2 17433.937} C_VEL
LIN {X 0,Y 390.556,Z 469.407,A -85,B 0,C 180,E1 17433.801,E2 17433.801} C_VEL
LIN {X 0,Y 393.616,Z 466.491,A -85,B 0,C 180,E1 17433.4,E2 17433.4} C_VEL
LIN {X 0,Y 396.755,Z 461.069,A -85,B 0,C 180,E1 17433.082,E2 17433.082} C_VEL
LIN {X 0,Y 400.709,Z 450.807,A -85,B 0,C 180,E1 17432.818,E2 17432.818} C_VEL
LIN {X 0,Y 403.114,Z 443.245,A -85,B 0,C 180,E1 17432.707,E2 17432.707} C_VEL
LIN {X 0,Y 406.902,Z 438.233,A -85,B 0,C 180,E1 17432.287,E2 17432.287} C_VEL
LIN {X 0,Y 410.768,Z 430.26,A -85,B 0,C 180,E1 17431.959,E2 17431.959} C_VEL
LIN {X 0,Y 412.711,Z 425.279,A -85,B 0,C 180,E1 17431.83,E2 17431.83} C_VEL
LIN {X 0,Y 408.607,Z 489.927,A -85,B 0,C 180,E1 17430.284,E2 17430.284} C_VEL
LIN {X 0,Y 406.971,Z 511.106,A -85,B 0,C 180,E1 17429.544,E2 17429.544} C_VEL
LIN {X 0,Y 404.822,Z 530.608,A -85,B 0,C 180,E1 17428.631,E2 17428.631} C_VEL
LIN {X 0,Y 402.048,Z 549.987,A -85,B 0,C 180,E1 17427.466,E2 17427.466} C_VEL
LIN {X 0,Y 398.84,Z 568.63,A -85,B 0,C 180,E1 17426.078,E2 17426.078} C_VEL
LIN {X 0,Y 395.04,Z 587.742,A -85,B 0,C 180,E1 17424.338,E2 17424.338} C_VEL
LIN {X 0,Y 391.16,Z 605.312,A -85,B 0,C 180,E1 17422.411,E2 17422.411} C_VEL
LIN {X 0,Y 387.303,Z 621.526,A -85,B 0,C 180,E1 17420.293,E2 17420.293} C_VEL
LIN {X 0,Y 383.306,Z 637.439,A -85,B 0,C 180,E1 17417.802,E2 17417.802} C_VEL
LIN {X 0,Y 379.718,Z 651.438,A -85,B 0,C 180,E1 17415.19,E2 17415.19} C_VEL
LIN {X 0,Y 376.548,Z 663.988,A -85,B 0,C 180,E1 17412.409,E2 17412.409} C_VEL
LIN {X 0,Y 373.785,Z 675.59,A -85,B 0,C 180,E1 17409.344,E2 17409.344} C_VEL
LIN {X 0,Y 372.662,Z 680.655,A -85,B 0,C 180,E1 17407.802,E2 17407.802} C_VEL
LIN {X 0,Y 370.987,Z 684.08,A -85,B 0,C 180,E1 17406.752,E2 17406.752} C_VEL
LIN {X 0,Y 363.651,Z 692.29,A -85,B 0,C 180,E1 17404.123,E2 17404.123} C_VEL
LIN {X 0,Y 362.192,Z 695.059,A -85,B 0,C 180,E1 17403.003,E2 17403.003} C_VEL
LIN {X 0,Y 361.109,Z 701.513,A -85,B 0,C 180,E1 17399.607,E2 17399.607} C_VEL
LIN {X 0,Y 360.509,Z 706.429,A -85,B 0,C 180,E1 17396.167,E2 17396.167} C_VEL
LIN {X 0,Y 360.247,Z 709.704,A -85,B 0,C 180,E1 17392.858,E2 17392.858} C_VEL
LIN {X 0,Y 360.141,Z 711.435,A -85,B 0,C 180,E1 17389.63,E2 17389.63} C_VEL
LIN {X 0,Y 360.129,Z 711.835,A -85,B 0,C 180,E1 17386.285,E2 17386.285} C_VEL
LIN {X 0,Y 360.164,Z 710.856,A -85,B 0,C 180,E1 17382.985,E2 17382.985} C_VEL
LIN {X 0,Y 360.303,Z 708.397,A -85,B 0,C 180,E1 17379.746,E2 17379.746} C_VEL
LIN {X 0,Y 360.699,Z 704.182,A -85,B 0,C 180,E1 17376.207,E2 17376.207} C_VEL
LIN {X 0,Y 361.46,Z 698.63,A -85,B 0,C 180,E1 17372.854,E2 17372.854} C_VEL
LIN {X 0,Y 362.701,Z 691.347,A -85,B 0,C 180,E1 17369.526,E2 17369.526} C_VEL
LIN {X 0,Y 364.441,Z 682.796,A -85,B 0,C 180,E1 17366.382,E2 17366.382} C_VEL
LIN {X 0,Y 366.803,Z 672.547,A -85,B 0,C 180,E1 17363.269,E2 17363.269} C_VEL
LIN {X 0,Y 369.662,Z 660.998,A -85,B 0,C 180,E1 17360.346,E2 17360.346} C_VEL
LIN {X 0,Y 373.137,Z 647.249,A -85,B 0,C 180,E1 17357.465,E2 17357.465} C_VEL
LIN {X 0,Y 376.766,Z 632.83,A -85,B 0,C 180,E1 17354.926,E2 17354.926} C_VEL
LIN {X 0,Y 380.656,Z 616.993,A -85,B 0,C 180,E1 17352.576,E2 17352.576} C_VEL
LIN {X 0,Y 384.415,Z 600.859,A -85,B 0,C 180,E1 17350.554,E2 17350.554} C_VEL
LIN {X 0,Y 388.333,Z 582.543,A -85,B 0,C 180,E1 17348.634,E2 17348.634} C_VEL
LIN {X 0,Y 391.862,Z 563.824,A -85,B 0,C 180,E1 17347.022,E2 17347.022} C_VEL
LIN {X 0,Y 394.881,Z 545.225,A -85,B 0,C 180,E1 17345.704,E2 17345.704} C_VEL
LIN {X 0,Y 397.494,Z 526.101,A -85,B 0,C 180,E1 17344.604,E2 17344.604} C_VEL
LIN {X 0,Y 399.702,Z 505.064,A -85,B 0,C 180,E1 17343.665,E2 17343.665} C_VEL
LIN {X 0,Y 401.175,Z 483.841,A -85,B 0,C 180,E1 17342.985,E2 17342.985} C_VEL
LIN {X 0,Y 409.755,Z 345.333,A -85,B 0,C 180,E1 17339.849,E2 17339.849} C_VEL
LIN {X 0,Y 413.839,Z 269.478,A -85,B 0,C 180,E1 17338.262,E2 17338.262} C_VEL
LIN {X 0,Y 400.609,Z 253.143,A -85,B 0,C 180,E1 17335.767,E2 17335.767} C_VEL
LIN {X 0,Y 387.503,Z 237.879,A -85,B 0,C 180,E1 17333.076,E2 17333.076} C_VEL
LIN {X 0,Y 381.737,Z 231.502,A -85,B 0,C 180,E1 17331.793,E2 17331.793} C_VEL
LIN {X 0,Y 379.307,Z 227.041,A -85,B 0,C 180,E1 17330.329,E2 17330.329} C_VEL
LIN {X 0,Y 377.008,Z 222.765,A -85,B 0,C 180,E1 17328.869,E2 17328.869} C_VEL
LIN {X 0,Y 374.266,Z 217.869,A -85,B 0,C 180,E1 17327.055,E2 17327.055} C_VEL
LIN {X 0,Y 371.94,Z 213.826,A -85,B 0,C 180,E1 17325.43,E2 17325.43} C_VEL
LIN {X 0,Y 368.894,Z 208.789,A -85,B 0,C 180,E1 17323.189,E2 17323.189} C_VEL
LIN {X 0,Y 368.218,Z 207.513,A -85,B 0,C 180,E1 17322.619,E2 17322.619} C_VEL
LIN {X 0,Y 365.831,Z 204.129,A -85,B 0,C 180,E1 17320.785,E2 17320.785} C_VEL
LIN {X 0,Y 365.078,Z 202.164,A -85,B 0,C 180,E1 17319.928,E2 17319.928} C_VEL
LIN {X 0,Y 362.44,Z 199,A -85,B 0,C 180,E1 17317.766,E2 17317.766} C_VEL
LIN {X 0,Y 361.794,Z 196.641,A -85,B 0,C 180,E1 17316.652,E2 17316.652} C_VEL
LIN {X 0,Y 361.774,Z 196.644,A -85,B 0,C 180,E1 17312.424,E2 17312.424} C_VEL
LIN {X 0,Y 361.79,Z 196.648,A -85,B 0,C 180,E1 17308.383,E2 17308.383} C_VEL
LIN {X 0,Y 361.801,Z 196.652,A -85,B 0,C 180,E1 17304.143,E2 17304.143} C_VEL
LIN {X 0,Y 361.806,Z 196.665,A -85,B 0,C 180,E1 17300.016,E2 17300.016} C_VEL
LIN {X 0,Y 361.772,Z 196.672,A -85,B 0,C 180,E1 17295.88,E2 17295.88} C_VEL
LIN {X 0,Y 361.752,Z 196.664,A -85,B 0,C 180,E1 17291.641,E2 17291.641} C_VEL
LIN {X 0,Y 361.781,Z 196.653,A -85,B 0,C 180,E1 17287.464,E2 17287.464} C_VEL
LIN {X 0,Y 361.8,Z 196.646,A -85,B 0,C 180,E1 17283.328,E2 17283.328} C_VEL
LIN {X 0,Y 361.807,Z 196.748,A -85,B 0,C 180,E1 17281.109,E2 17281.109} C_VEL
LIN {X 0,Y 363.314,Z 200.447,A -85,B 0,C 180,E1 17279.212,E2 17279.212} C_VEL
LIN {X 0,Y 365.358,Z 202.701,A -85,B 0,C 180,E1 17277.648,E2 17277.648} C_VEL
LIN {X 0,Y 367.153,Z 206.434,A -85,B 0,C 180,E1 17275.94,E2 17275.94} C_VEL
LIN {X 0,Y 368.708,Z 208.307,A -85,B 0,C 180,E1 17274.866,E2 17274.866} C_VEL
LIN {X 0,Y 370.56,Z 212.003,A -85,B 0,C 180,E1 17273.338,E2 17273.338} C_VEL
LIN {X 0,Y 371.761,Z 213.545,A -85,B 0,C 180,E1 17272.583,E2 17272.583} C_VEL
LIN {X 0,Y 373.884,Z 217.453,A -85,B 0,C 180,E1 17271.078,E2 17271.078} C_VEL
LIN {X 0,Y 375.022,Z 219.393,A -85,B 0,C 180,E1 17270.331,E2 17270.331} C_VEL
LIN {X 0,Y 377.796,Z 224.327,A -85,B 0,C 180,E1 17268.552,E2 17268.552} C_VEL
LIN {X 0,Y 382.556,Z 232.771,A -85,B 0,C 180,E1 17265.778,E2 17265.778} C_VEL
LIN {X 0,Y 389.318,Z 246.012,A -85,B 0,C 180,E1 17262.05,E2 17262.05} C_VEL
LIN {X 0,Y 395.95,Z 259.926,A -85,B 0,C 180,E1 17258.677,E2 17258.677} C_VEL
LIN {X 0,Y 402.282,Z 274.085,A -85,B 0,C 180,E1 17255.633,E2 17255.633} C_VEL
LIN {X 0,Y 408.759,Z 289.532,A -85,B 0,C 180,E1 17252.658,E2 17252.658} C_VEL
LIN {X 0,Y 402.767,Z 333.2,A -85,B 0,C 180,E1 17248.496,E2 17248.496} C_VEL
LIN {X 0,Y 402.064,Z 353.66,A -85,B 0,C 180,E1 17246.32,E2 17246.32} C_VEL
LIN {X 0,Y 403.38,Z 372.241,A -85,B 0,C 180,E1 17244.148,E2 17244.148} C_VEL
LIN {X 0,Y 406.909,Z 390.379,A -85,B 0,C 180,E1 17241.841,E2 17241.841} C_VEL
LIN {X 0,Y 412.295,Z 406.353,A -85,B 0,C 180,E1 17239.647,E2 17239.647} C_VEL
LIN {X 0,Y 419.808,Z 421.355,A -85,B 0,C 180,E1 17237.437,E2 17237.437} C_VEL
LIN {X 0,Y 423.415,Z 427.164,A -85,B 0,C 180,E1 17236.548,E2 17236.548} C_VEL
LIN {X 0,Y 413.27,Z 445.033,A -85,B 0,C 180,E1 17235.816,E2 17235.816} C_VEL
LIN {X 0,Y 408.347,Z 474.879,A -85,B 0,C 180,E1 17235.751,E2 17235.751} C_VEL
LIN {X 0,Y 405.795,Z 496.509,A -85,B 0,C 180,E1 17235.455,E2 17235.455} C_VEL
LIN {X 0,Y 403.039,Z 523.742,A -85,B 0,C 180,E1 17234.686,E2 17234.686} C_VEL
LIN {X 0,Y 399.408,Z 549.834,A -85,B 0,C 180,E1 17233.728,E2 17233.728} C_VEL
LIN {X 0,Y 395.519,Z 574.284,A -85,B 0,C 180,E1 17232.542,E2 17232.542} C_VEL
LIN {X 0,Y 391.483,Z 597.601,A -85,B 0,C 180,E1 17231.111,E2 17231.111} C_VEL
LIN {X 0,Y 387.301,Z 620.032,A -85,B 0,C 180,E1 17229.425,E2 17229.425} C_VEL
LIN {X 0,Y 383.381,Z 640.14,A -85,B 0,C 180,E1 17227.609,E2 17227.609} C_VEL
LIN {X 0,Y 379.568,Z 658.938,A -85,B 0,C 180,E1 17225.602,E2 17225.602} C_VEL
LIN {X 0,Y 375.558,Z 677.795,A -85,B 0,C 180,E1 17223.178,E2 17223.178} C_VEL
LIN {X 0,Y 372.003,Z 694.108,A -85,B 0,C 180,E1 17220.674,E2 17220.674} C_VEL
LIN {X 0,Y 368.836,Z 709.096,A -85,B 0,C 180,E1 17217.968,E2 17217.968} C_VEL
LIN {X 0,Y 365.935,Z 723.328,A -85,B 0,C 180,E1 17214.884,E2 17214.884} C_VEL
LIN {X 0,Y 363.826,Z 734.711,A -85,B 0,C 180,E1 17211.947,E2 17211.947} C_VEL
LIN {X 0,Y 362.059,Z 745.712,A -85,B 0,C 180,E1 17208.517,E2 17208.517} C_VEL
LIN {X 0,Y 360.942,Z 754.469,A -85,B 0,C 180,E1 17205.093,E2 17205.093} C_VEL
LIN {X 0,Y 360.366,Z 761.025,A -85,B 0,C 180,E1 17201.848,E2 17201.848} C_VEL
LIN {X 0,Y 360.118,Z 766.07,A -85,B 0,C 180,E1 17198.462,E2 17198.462} C_VEL
LIN {X 0,Y 360.085,Z 769.29,A -85,B 0,C 180,E1 17195.257,E2 17195.257} C_VEL
LIN {X 0,Y 360.11,Z 770.934,A -85,B 0,C 180,E1 17192.068,E2 17192.068} C_VEL
LIN {X 0,Y 360.121,Z 771.115,A -85,B 0,C 180,E1 17188.886,E2 17188.886} C_VEL
LIN {X 0,Y 360.1,Z 769.794,A -85,B 0,C 180,E1 17185.7,E2 17185.7} C_VEL
LIN {X 0,Y 360.109,Z 766.77,A -85,B 0,C 180,E1 17182.341,E2 17182.341} C_VEL
LIN {X 0,Y 360.276,Z 762.298,A -85,B 0,C 180,E1 17179.122,E2 17179.122} C_VEL
LIN {X 0,Y 360.763,Z 755.8,A -85,B 0,C 180,E1 17175.719,E2 17175.719} C_VEL
LIN {X 0,Y 361.668,Z 747.854,A -85,B 0,C 180,E1 17172.462,E2 17172.462} C_VEL
LIN {X 0,Y 363.22,Z 737.424,A -85,B 0,C 180,E1 17169.031,E2 17169.031} C_VEL
LIN {X 0,Y 365.236,Z 725.984,A -85,B 0,C 180,E1 17165.927,E2 17165.927} C_VEL
LIN {X 0,Y 367.937,Z 712.352,A -85,B 0,C 180,E1 17162.836,E2 17162.836} C_VEL
LIN {X 0,Y 371.18,Z 697.087,A -85,B 0,C 180,E1 17159.931,E2 17159.931} C_VEL
LIN {X 0,Y 374.776,Z 680.65,A -85,B 0,C 180,E1 17157.299,E2 17157.299} C_VEL
LIN {X 0,Y 378.714,Z 662.571,A -85,B 0,C 180,E1 17154.861,E2 17154.861} C_VEL
LIN {X 0,Y 382.784,Z 643.373,A -85,B 0,C 180,E1 17152.699,E2 17152.699} C_VEL
LIN {X 0,Y 387.345,Z 620.559,A -85,B 0,C 180,E1 17150.579,E2 17150.579} C_VEL
LIN {X 0,Y 391.574,Z 598.554,A -85,B 0,C 180,E1 17148.889,E2 17148.889} C_VEL
LIN {X 0,Y 395.858,Z 574.814,A -85,B 0,C 180,E1 17147.396,E2 17147.396} C_VEL
LIN {X 0,Y 399.986,Z 550.705,A -85,B 0,C 180,E1 17146.177,E2 17146.177} C_VEL
LIN {X 0,Y 403.948,Z 524.675,A -85,B 0,C 180,E1 17145.171,E2 17145.171} C_VEL
LIN {X 0,Y 407.123,Z 497.285,A -85,B 0,C 180,E1 17144.346,E2 17144.346} C_VEL
LIN {X 0,Y 409.955,Z 472.441,A -85,B 0,C 180,E1 17143.905,E2 17143.905} C_VEL
LIN {X 0,Y 414.224,Z 435.776,A -85,B 0,C 180,E1 17143.638,E2 17143.638} C_VEL
LIN {X 0,Y 415.067,Z 430.143,A -85,B 0,C 180,E1 17143.624,E2 17143.624} C_VEL
LIN {X 0,Y 419.917,Z 417.057,A -85,B 0,C 180,E1 17143.229,E2 17143.229} C_VEL
LIN {X 0,Y 427.69,Z 395.58,A -85,B 0,C 180,E1 17142.573,E2 17142.573} C_VEL
LIN {X 0,Y 438.145,Z 370.947,A -85,B 0,C 180,E1 17142.029,E2 17142.029} C_VEL
LIN {X 0,Y 447.13,Z 351.567,A -85,B 0,C 180,E1 17141.708,E2 17141.708} C_VEL
LIN {X 0,Y 437.888,Z 338.687,A -85,B 0,C 180,E1 17139.572,E2 17139.572} C_VEL
LIN {X 0,Y 430.85,Z 324.562,A -85,B 0,C 180,E1 17137.446,E2 17137.446} C_VEL
LIN {X 0,Y 428.541,Z 318.622,A -85,B 0,C 180,E1 17136.591,E2 17136.591} C_VEL
LIN {X 0,Y 413.388,Z 328.607,A -85,B 0,C 180,E1 17134.975,E2 17134.975} C_VEL
LIN {X 0,Y 406.95,Z 333.024,A -85,B 0,C 180,E1 17134.238,E2 17134.238} C_VEL
LIN {X 0,Y 401.441,Z 336.742,A -85,B 0,C 180,E1 17133.568,E2 17133.568} C_VEL
LIN {X 0,Y 397.333,Z 339.993,A -85,B 0,C 180,E1 17133.097,E2 17133.097} C_VEL
LIN {X 0,Y 394.599,Z 341.695,A -85,B 0,C 180,E1 17132.728,E2 17132.728} C_VEL
LIN {X 0,Y 390.968,Z 344.757,A -85,B 0,C 180,E1 17132.309,E2 17132.309} C_VEL
LIN {X 0,Y 388.446,Z 346.122,A -85,B 0,C 180,E1 17131.891,E2 17131.891} C_VEL
LIN {X 0,Y 387.883,Z 353.111,A -85,B 0,C 180,E1 17131.206,E2 17131.206} C_VEL
LIN {X 0,Y 384.518,Z 366.022,A -85,B 0,C 180,E1 17130.43,E2 17130.43} C_VEL
LIN {X 0,Y 377.567,Z 462.512,A -85,B 0,C 180,E1 17127.571,E2 17127.571} C_VEL
LIN {X 0,Y 375.311,Z 511.408,A -85,B 0,C 180,E1 17126.174,E2 17126.174} C_VEL
LIN {X 0,Y 374.995,Z 533.066,A -85,B 0,C 180,E1 17125.442,E2 17125.442} C_VEL
LIN {X 0,Y 374.446,Z 550.531,A -85,B 0,C 180,E1 17124.575,E2 17124.575} C_VEL
LIN {X 0,Y 373.547,Z 567.664,A -85,B 0,C 180,E1 17123.421,E2 17123.421} C_VEL
LIN {X 0,Y 372.432,Z 583.048,A -85,B 0,C 180,E1 17122.077,E2 17122.077} C_VEL
LIN {X 0,Y 371.128,Z 597.358,A -85,B 0,C 180,E1 17120.501,E2 17120.501} C_VEL
LIN {X 0,Y 369.754,Z 609.979,A -85,B 0,C 180,E1 17118.771,E2 17118.771} C_VEL
LIN {X 0,Y 368.362,Z 621.082,A -85,B 0,C 180,E1 17116.883,E2 17116.883} C_VEL
LIN {X 0,Y 367.007,Z 630.723,A -85,B 0,C 180,E1 17114.838,E2 17114.838} C_VEL
LIN {X 0,Y 365.765,Z 639.085,A -85,B 0,C 180,E1 17112.603,E2 17112.603} C_VEL
LIN {X 0,Y 364.699,Z 645.739,A -85,B 0,C 180,E1 17110.265,E2 17110.265} C_VEL
LIN {X 0,Y 363.775,Z 650.885,A -85,B 0,C 180,E1 17107.74,E2 17107.74} C_VEL
LIN {X 0,Y 363.113,Z 654.204,A -85,B 0,C 180,E1 17105.213,E2 17105.213} C_VEL
LIN {X 0,Y 362.667,Z 655.785,A -85,B 0,C 180,E1 17102.686,E2 17102.686} C_VEL
LIN {X 0,Y 362.392,Z 655.644,A -85,B 0,C 180,E1 17100.158,E2 17100.158} C_VEL
LIN {X 0,Y 362.263,Z 653.71,A -85,B 0,C 180,E1 17097.468,E2 17097.468} C_VEL
LIN {X 0,Y 362.322,Z 650.194,A -85,B 0,C 180,E1 17094.933,E2 17094.933} C_VEL
LIN {X 0,Y 362.567,Z 644.877,A -85,B 0,C 180,E1 17092.393,E2 17092.393} C_VEL
LIN {X 0,Y 363.05,Z 637.648,A -85,B 0,C 180,E1 17089.847,E2 17089.847} C_VEL
LIN {X 0,Y 363.727,Z 628.903,A -85,B 0,C 180,E1 17087.457,E2 17087.457} C_VEL
LIN {X 0,Y 364.594,Z 618.611,A -85,B 0,C 180,E1 17085.223,E2 17085.223} C_VEL
LIN {X 0,Y 365.677,Z 606.393,A -85,B 0,C 180,E1 17083.07,E2 17083.07} C_VEL
LIN {X 0,Y 366.828,Z 593.008,A -85,B 0,C 180,E1 17081.155,E2 17081.155} C_VEL
LIN {X 0,Y 368.034,Z 577.835,A -85,B 0,C 180,E1 17079.401,E2 17079.401} C_VEL
LIN {X 0,Y 369.122,Z 562.467,A -85,B 0,C 180,E1 17077.965,E2 17077.965} C_VEL
LIN {X 0,Y 370.101,Z 545.305,A -85,B 0,C 180,E1 17076.714,E2 17076.714} C_VEL
LIN {X 0,Y 370.883,Z 526.998,A -85,B 0,C 180,E1 17075.706,E2 17075.706} C_VEL
LIN {X 0,Y 371.28,Z 514.224,A -85,B 0,C 180,E1 17075.179,E2 17075.179} C_VEL
LIN {X 0,Y 372.369,Z 515.379,A -85,B 0,C 180,E1 17074.896,E2 17074.896} C_VEL
LIN {X 0,Y 374.078,Z 514.78,A -85,B 0,C 180,E1 17074.613,E2 17074.613} C_VEL
LIN {X 0,Y 376.737,Z 511.667,A -85,B 0,C 180,E1 17074.314,E2 17074.314} C_VEL
LIN {X 0,Y 380.216,Z 504.596,A -85,B 0,C 180,E1 17074.086,E2 17074.086} C_VEL
LIN {X 0,Y 382.155,Z 499.085,A -85,B 0,C 180,E1 17074.008,E2 17074.008} C_VEL
LIN {X 0,Y 385.286,Z 496.249,A -85,B 0,C 180,E1 17073.599,E2 17073.599} C_VEL
LIN {X 0,Y 388.575,Z 490.831,A -85,B 0,C 180,E1 17073.282,E2 17073.282} C_VEL
LIN {X 0,Y 392.507,Z 480.896,A -85,B 0,C 180,E1 17073.025,E2 17073.025} C_VEL
LIN {X 0,Y 394.717,Z 474.22,A -85,B 0,C 180,E1 17072.918,E2 17072.918} C_VEL
LIN {X 0,Y 398.556,Z 469.306,A -85,B 0,C 180,E1 17072.487,E2 17072.487} C_VEL
LIN {X 0,Y 402.495,Z 461.479,A -85,B 0,C 180,E1 17072.158,E2 17072.158} C_VEL
LIN {X 0,Y 405.28,Z 454.223,A -85,B 0,C 180,E1 17071.982,E2 17071.982} C_VEL
LIN {X 0,Y 402.626,Z 494.461,A -85,B 0,C 180,E1 17070.949,E2 17070.949} C_VEL
LIN {X 0,Y 400.833,Z 515.235,A -85,B 0,C 180,E1 17070.176,E2 17070.176} C_VEL
LIN {X 0,Y 398.308,Z 535.859,A -85,B 0,C 180,E1 17069.15,E2 17069.15} C_VEL
LIN {X 0,Y 395.316,Z 555.236,A -85,B 0,C 180,E1 17067.916,E2 17067.916} C_VEL
LIN {X 0,Y 391.788,Z 574.206,A -85,B 0,C 180,E1 17066.421,E2 17066.421} C_VEL
LIN {X 0,Y 387.915,Z 592.294,A -85,B 0,C 180,E1 17064.678,E2 17064.678} C_VEL
LIN {X 0,Y 383.883,Z 609.249,A -85,B 0,C 180,E1 17062.722,E2 17062.722} C_VEL
LIN {X 0,Y 379.603,Z 626.066,A -85,B 0,C 180,E1 17060.4,E2 17060.4} C_VEL
LIN {X 0,Y 375.654,Z 640.946,A -85,B 0,C 180,E1 17057.954,E2 17057.954} C_VEL
LIN {X 0,Y 371.893,Z 654.935,A -85,B 0,C 180,E1 17055.218,E2 17055.218} C_VEL
LIN {X 0,Y 368.37,Z 668.182,A -85,B 0,C 180,E1 17052.101,E2 17052.101} C_VEL
LIN {X 0,Y 365.611,Z 679.114,A -85,B 0,C 180,E1 17048.976,E2 17048.976} C_VEL
LIN {X 0,Y 363.438,Z 688.632,A -85,B 0,C 180,E1 17045.679,E2 17045.679} C_VEL
LIN {X 0,Y 362.192,Z 695.059,A -85,B 0,C 180,E1 17043.003,E2 17043.003} C_VEL
LIN {X 0,Y 360.784,Z 697.654,A -85,B 0,C 180,E1 17041.865,E2 17041.865} C_VEL
LIN {X 0,Y 353.736,Z 703.849,A -85,B 0,C 180,E1 17038.799,E2 17038.799} C_VEL
LIN {X 0,Y 352.794,Z 705.402,A -85,B 0,C 180,E1 17037.757,E2 17037.757} C_VEL
LIN {X 0,Y 352.377,Z 709.266,A -85,B 0,C 180,E1 17034.295,E2 17034.295} C_VEL
LIN {X 0,Y 352.2,Z 711.637,A -85,B 0,C 180,E1 17030.932,E2 17030.932} C_VEL
LIN {X 0,Y 352.152,Z 712.506,A -85,B 0,C 180,E1 17027.686,E2 17027.686} C_VEL
LIN {X 0,Y 352.174,Z 712.057,A -85,B 0,C 180,E1 17024.301,E2 17024.301} C_VEL
LIN {X 0,Y 352.273,Z 710.187,A -85,B 0,C 180,E1 17020.868,E2 17020.868} C_VEL
LIN {X 0,Y 352.557,Z 706.791,A -85,B 0,C 180,E1 17017.496,E2 17017.496} C_VEL
LIN {X 0,Y 353.213,Z 701.579,A -85,B 0,C 180,E1 17013.896,E2 17013.896} C_VEL
LIN {X 0,Y 354.359,Z 695.005,A -85,B 0,C 180,E1 17010.485,E2 17010.485} C_VEL
LIN {X 0,Y 356.164,Z 686.285,A -85,B 0,C 180,E1 17006.943,E2 17006.943} C_VEL
LIN {X 0,Y 358.589,Z 675.967,A -85,B 0,C 180,E1 17003.597,E2 17003.597} C_VEL
LIN {X 0,Y 361.428,Z 664.806,A -85,B 0,C 180,E1 17000.606,E2 17000.606} C_VEL
LIN {X 0,Y 364.905,Z 651.679,A -85,B 0,C 180,E1 16997.66,E2 16997.66} C_VEL
LIN {X 0,Y 368.584,Z 637.922,A -85,B 0,C 180,E1 16995.066,E2 16995.066} C_VEL
LIN {X 0,Y 372.499,Z 622.802,A -85,B 0,C 180,E1 16992.666,E2 16992.666} C_VEL
LIN {X 0,Y 376.437,Z 606.766,A -85,B 0,C 180,E1 16990.528,E2 16990.528} C_VEL
LIN {X 0,Y 380.413,Z 589.321,A -85,B 0,C 180,E1 16988.572,E2 16988.572} C_VEL
LIN {X 0,Y 384.169,Z 570.997,A -85,B 0,C 180,E1 16986.859,E2 16986.859} C_VEL
LIN {X 0,Y 387.624,Z 551.762,A -85,B 0,C 180,E1 16985.381,E2 16985.381} C_VEL
LIN {X 0,Y 390.461,Z 532.475,A -85,B 0,C 180,E1 16984.194,E2 16984.194} C_VEL
LIN {X 0,Y 392.868,Z 512.057,A -85,B 0,C 180,E1 16983.206,E2 16983.206} C_VEL
LIN {X 0,Y 394.63,Z 491.161,A -85,B 0,C 180,E1 16982.448,E2 16982.448} C_VEL
LIN {X 0,Y 398.354,Z 432.995,A -85,B 0,C 180,E1 16981.02,E2 16981.02} C_VEL
LIN {X 0,Y 405.626,Z 320.133,A -85,B 0,C 180,E1 16978.506,E2 16978.506} C_VEL
LIN {X 0,Y 408.083,Z 273.474,A -85,B 0,C 180,E1 16977.512,E2 16977.512} C_VEL
LIN {X 0,Y 393.959,Z 255.988,A -85,B 0,C 180,E1 16974.746,E2 16974.746} C_VEL
LIN {X 0,Y 379.89,Z 239.793,A -85,B 0,C 180,E1 16971.72,E2 16971.72} C_VEL
LIN {X 0,Y 375.537,Z 234.921,A -85,B 0,C 180,E1 16970.679,E2 16970.679} C_VEL
LIN {X 0,Y 371.853,Z 228.431,A -85,B 0,C 180,E1 16968.375,E2 16968.375} C_VEL
LIN {X 0,Y 369.443,Z 224.032,A -85,B 0,C 180,E1 16966.722,E2 16966.722} C_VEL
LIN {X 0,Y 366.679,Z 219.136,A -85,B 0,C 180,E1 16964.71,E2 16964.71} C_VEL
LIN {X 0,Y 364.522,Z 215.588,A -85,B 0,C 180,E1 16963.078,E2 16963.078} C_VEL
LIN {X 0,Y 363.934,Z 214.243,A -85,B 0,C 180,E1 16962.521,E2 16962.521} C_VEL
LIN {X 0,Y 361.431,Z 210.645,A -85,B 0,C 180,E1 16960.55,E2 16960.55} C_VEL
LIN {X 0,Y 360.817,Z 208.918,A -85,B 0,C 180,E1 16959.802,E2 16959.802} C_VEL
LIN {X 0,Y 358.112,Z 205.514,A -85,B 0,C 180,E1 16957.494,E2 16957.494} C_VEL
LIN {X 0,Y 357.358,Z 203.306,A -85,B 0,C 180,E1 16956.382,E2 16956.382} C_VEL
LIN {X 0,Y 354.476,Z 199.981,A -85,B 0,C 180,E1 16953.37,E2 16953.37} C_VEL
LIN {X 0,Y 353.816,Z 197.634,A -85,B 0,C 180,E1 16951.901,E2 16951.901} C_VEL
LIN {X 0,Y 353.844,Z 197.631,A -85,B 0,C 180,E1 16947.791,E2 16947.791} C_VEL
LIN {X 0,Y 353.866,Z 197.632,A -85,B 0,C 180,E1 16943.655,E2 16943.655} C_VEL
LIN {X 0,Y 353.848,Z 197.642,A -85,B 0,C 180,E1 16939.478,E2 16939.478} C_VEL
LIN {X 0,Y 353.823,Z 197.656,A -85,B 0,C 180,E1 16935.237,E2 16935.237} C_VEL
LIN {X 0,Y 353.843,Z 197.661,A -85,B 0,C 180,E1 16930.914,E2 16930.914} C_VEL
LIN {X 0,Y 353.875,Z 197.654,A -85,B 0,C 180,E1 16926.653,E2 16926.653} C_VEL
LIN {X 0,Y 353.851,Z 197.656,A -85,B 0,C 180,E1 16925.839,E2 16925.839} C_VEL
LIN {X 0,Y 355.587,Z 201.687,A -85,B 0,C 180,E1 16923.063,E2 16923.063} C_VEL
LIN {X 0,Y 357.54,Z 203.531,A -85,B 0,C 180,E1 16921.282,E2 16921.282} C_VEL
LIN {X 0,Y 359.244,Z 207.397,A -85,B 0,C 180,E1 16919.203,E2 16919.203} C_VEL
LIN {X 0,Y 360.915,Z 209.11,A -85,B 0,C 180,E1 16917.937,E2 16917.937} C_VEL
LIN {X 0,Y 362.87,Z 213.157,A -85,B 0,C 180,E1 16916.051,E2 16916.051} C_VEL
LIN {X 0,Y 364.194,Z 214.746,A -85,B 0,C 180,E1 16915.118,E2 16915.118} C_VEL
LIN {X 0,Y 366.007,Z 218.437,A -85,B 0,C 180,E1 16913.57,E2 16913.57} C_VEL
LIN {X 0,Y 367.18,Z 219.995,A -85,B 0,C 180,E1 16912.805,E2 16912.805} C_VEL
LIN {X 0,Y 369.549,Z 224.195,A -85,B 0,C 180,E1 16911.129,E2 16911.129} C_VEL
LIN {X 0,Y 373.138,Z 230.798,A -85,B 0,C 180,E1 16908.72,E2 16908.72} C_VEL
LIN {X 0,Y 377.809,Z 239.322,A -85,B 0,C 180,E1 16905.909,E2 16905.909} C_VEL
LIN {X 0,Y 383.434,Z 250.489,A -85,B 0,C 180,E1 16902.707,E2 16902.707} C_VEL
LIN {X 0,Y 389.453,Z 262.938,A -85,B 0,C 180,E1 16899.565,E2 16899.565} C_VEL
LIN {X 0,Y 395.935,Z 277.508,A -85,B 0,C 180,E1 16896.327,E2 16896.327} C_VEL
LIN {X 0,Y 402.529,Z 293.461,A -85,B 0,C 180,E1 16893.181,E2 16893.181} C_VEL
LIN {X 0,Y 396.428,Z 336.368,A -85,B 0,C 180,E1 16889.041,E2 16889.041} C_VEL
LIN {X 0,Y 395.631,Z 357.586,A -85,B 0,C 180,E1 16886.742,E2 16886.742} C_VEL
LIN {X 0,Y 396.951,Z 376.423,A -85,B 0,C 180,E1 16884.499,E2 16884.499} C_VEL
LIN {X 0,Y 400.523,Z 394.855,A -85,B 0,C 180,E1 16882.113,E2 16882.113} C_VEL
LIN {X 0,Y 406.047,Z 411.228,A -85,B 0,C 180,E1 16879.823,E2 16879.823} C_VEL
LIN {X 0,Y 413.555,Z 426.232,A -85,B 0,C 180,E1 16877.582,E2 16877.582} C_VEL
LIN {X 0,Y 415.219,Z 429.356,A -85,B 0,C 180,E1 16877.119,E2 16877.119} C_VEL
LIN {X 0,Y 407.852,Z 442.688,A -85,B 0,C 180,E1 16876.586,E2 16876.586} C_VEL
LIN {X 0,Y 402.8,Z 472.542,A -85,B 0,C 180,E1 16876.541,E2 16876.541} C_VEL
LIN {X 0,Y 399.994,Z 494.863,A -85,B 0,C 180,E1 16876.247,E2 16876.247} C_VEL
LIN {X 0,Y 397.187,Z 521.495,A -85,B 0,C 180,E1 16875.498,E2 16875.498} C_VEL
LIN {X 0,Y 393.462,Z 547.65,A -85,B 0,C 180,E1 16874.537,E2 16874.537} C_VEL
LIN {X 0,Y 389.365,Z 572.364,A -85,B 0,C 180,E1 16873.341,E2 16873.341} C_VEL
LIN {X 0,Y 385.061,Z 596.409,A -85,B 0,C 180,E1 16871.861,E2 16871.861} C_VEL
LIN {X 0,Y 380.729,Z 618.952,A -85,B 0,C 180,E1 16870.163,E2 16870.163} C_VEL
LIN {X 0,Y 376.451,Z 640.185,A -85,B 0,C 180,E1 16868.232,E2 16868.232} C_VEL
LIN {X 0,Y 372.472,Z 658.792,A -85,B 0,C 180,E1 16866.197,E2 16866.197} C_VEL
LIN {X 0,Y 368.404,Z 677.19,A -85,B 0,C 180,E1 16863.805,E2 16863.805} C_VEL
LIN {X 0,Y 364.407,Z 694.766,A -85,B 0,C 180,E1 16861.053,E2 16861.053} C_VEL
LIN {X 0,Y 361.124,Z 709.465,A -85,B 0,C 180,E1 16858.303,E2 16858.303} C_VEL
LIN {X 0,Y 358.212,Z 723.199,A -85,B 0,C 180,E1 16855.263,E2 16855.263} C_VEL
LIN {X 0,Y 355.9,Z 735.005,A -85,B 0,C 180,E1 16852.114,E2 16852.114} C_VEL
LIN {X 0,Y 354.223,Z 744.926,A -85,B 0,C 180,E1 16848.942,E2 16848.942} C_VEL
LIN {X 0,Y 353.024,Z 753.735,A -85,B 0,C 180,E1 16845.44,E2 16845.44} C_VEL
LIN {X 0,Y 352.399,Z 760.322,A -85,B 0,C 180,E1 16842.12,E2 16842.12} C_VEL
LIN {X 0,Y 352.135,Z 765.391,A -85,B 0,C 180,E1 16838.655,E2 16838.655} C_VEL
LIN {X 0,Y 352.106,Z 768.623,A -85,B 0,C 180,E1 16835.377,E2 16835.377} C_VEL
LIN {X 0,Y 352.136,Z 770.274,A -85,B 0,C 180,E1 16832.115,E2 16832.115} C_VEL
LIN {X 0,Y 352.147,Z 770.456,A -85,B 0,C 180,E1 16828.861,E2 16828.861} C_VEL
LIN {X 0,Y 352.122,Z 769.138,A -85,B 0,C 180,E1 16825.603,E2 16825.603} C_VEL
LIN {X 0,Y 352.129,Z 766.094,A -85,B 0,C 180,E1 16822.166,E2 16822.166} C_VEL
LIN {X 0,Y 352.301,Z 761.629,A -85,B 0,C 180,E1 16818.872,E2 16818.872} C_VEL
LIN {X 0,Y 352.827,Z 755.121,A -85,B 0,C 180,E1 16815.391,E2 16815.391} C_VEL
LIN {X 0,Y 353.798,Z 747.169,A -85,B 0,C 180,E1 16812.058,E2 16812.058} C_VEL
LIN {X 0,Y 355.471,Z 736.732,A -85,B 0,C 180,E1 16808.551,E2 16808.551} C_VEL
LIN {X 0,Y 357.704,Z 724.92,A -85,B 0,C 180,E1 16805.29,E2 16805.29} C_VEL
LIN {X 0,Y 360.532,Z 711.577,A -85,B 0,C 180,E1 16802.211,E2 16802.211} C_VEL
LIN {X 0,Y 363.904,Z 696.632,A -85,B 0,C 180,E1 16799.315,E2 16799.315} C_VEL
LIN {X 0,Y 367.658,Z 680.513,A -85,B 0,C 180,E1 16796.677,E2 16796.677} C_VEL
LIN {X 0,Y 371.656,Z 663.146,A -85,B 0,C 180,E1 16794.282,E2 16794.282} C_VEL
LIN {X 0,Y 375.914,Z 644.209,A -85,B 0,C 180,E1 16792.09,E2 16792.09} C_VEL
LIN {X 0,Y 380.086,Z 624.385,A -85,B 0,C 180,E1 16790.186,E2 16790.186} C_VEL
LIN {X 0,Y 384.837,Z 600.92,A -85,B 0,C 180,E1 16788.308,E2 16788.308} C_VEL
LIN {X 0,Y 389.264,Z 578.009,A -85,B 0,C 180,E1 16786.801,E2 16786.801} C_VEL
LIN {X 0,Y 393.691,Z 553.039,A -85,B 0,C 180,E1 16785.496,E2 16785.496} C_VEL
LIN {X 0,Y 398.027,Z 526.215,A -85,B 0,C 180,E1 16784.419,E2 16784.419} C_VEL
LIN {X 0,Y 401.552,Z 498.194,A -85,B 0,C 180,E1 16783.539,E2 16783.539} C_VEL
LIN {X 0,Y 404.407,Z 474.818,A -85,B 0,C 180,E1 16783.089,E2 16783.089} C_VEL
LIN {X 0,Y 408.907,Z 436.475,A -85,B 0,C 180,E1 16782.791,E2 16782.791} C_VEL
LIN {X 0,Y 410.587,Z 426.128,A -85,B 0,C 180,E1 16782.759,E2 16782.759} C_VEL
LIN {X 0,Y 414.933,Z 414.193,A -85,B 0,C 180,E1 16782.39,E2 16782.39} C_VEL
LIN {X 0,Y 423.366,Z 391.562,A -85,B 0,C 180,E1 16781.729,E2 16781.729} C_VEL
LIN {X 0,Y 434.54,Z 365.786,A -85,B 0,C 180,E1 16781.2,E2 16781.2} C_VEL
LIN {X 0,Y 439.633,Z 354.565,A -85,B 0,C 180,E1 16781.004,E2 16781.004} C_VEL
LIN {X 0,Y 431.275,Z 342.004,A -85,B 0,C 180,E1 16778.923,E2 16778.923} C_VEL
LIN {X 0,Y 424.618,Z 328.013,A -85,B 0,C 180,E1 16776.776,E2 16776.776} C_VEL
LIN {X 0,Y 413.71,Z 335.12,A -85,B 0,C 180,E1 16775.623,E2 16775.623} C_VEL
LIN {X 0,Y 407.173,Z 339.545,A -85,B 0,C 180,E1 16774.9,E2 16774.9} C_VEL
LIN {X 0,Y 401.564,Z 343.4,A -85,B 0,C 180,E1 16774.244,E2 16774.244} C_VEL
LIN {X 0,Y 396.099,Z 347.288,A -85,B 0,C 180,E1 16773.59,E2 16773.59} C_VEL
LIN {X 0,Y 390.299,Z 351.691,A -85,B 0,C 180,E1 16772.894,E2 16772.894} C_VEL
LIN {X 0,Y 388.85,Z 352.465,A -85,B 0,C 180,E1 16772.682,E2 16772.682} C_VEL
LIN {X 0,Y 382.175,Z 358.333,A -85,B 0,C 180,E1 16771.902,E2 16771.902} C_VEL
LIN {X 0,Y 381.426,Z 358.926,A -85,B 0,C 180,E1 16771.795,E2 16771.795} C_VEL
LIN {X 0,Y 378.869,Z 368.633,A -85,B 0,C 180,E1 16771.238,E2 16771.238} C_VEL
LIN {X 0,Y 371.414,Z 461.258,A -85,B 0,C 180,E1 16768.379,E2 16768.379} C_VEL
LIN {X 0,Y 368.718,Z 510.909,A -85,B 0,C 180,E1 16766.892,E2 16766.892} C_VEL
LIN {X 0,Y 368.244,Z 534.214,A -85,B 0,C 180,E1 16766.081,E2 16766.081} C_VEL
LIN {X 0,Y 367.606,Z 552.552,A -85,B 0,C 180,E1 16765.149,E2 16765.149} C_VEL
LIN {X 0,Y 366.608,Z 569.42,A -85,B 0,C 180,E1 16763.977,E2 16763.977} C_VEL
LIN {X 0,Y 365.416,Z 584.799,A -85,B 0,C 180,E1 16762.608,E2 16762.608} C_VEL
LIN {X 0,Y 363.997,Z 599,A -85,B 0,C 180,E1 16761.006,E2 16761.006} C_VEL
LIN {X 0,Y 362.465,Z 612.162,A -85,B 0,C 180,E1 16759.163,E2 16759.163} C_VEL
LIN {X 0,Y 360.96,Z 623.102,A -85,B 0,C 180,E1 16757.24,E2 16757.24} C_VEL
LIN {X 0,Y 359.415,Z 633.342,A -85,B 0,C 180,E1 16754.993,E2 16754.993} C_VEL
LIN {X 0,Y 358.104,Z 641.359,A -85,B 0,C 180,E1 16752.742,E2 16752.742} C_VEL
LIN {X 0,Y 356.876,Z 648.227,A -85,B 0,C 180,E1 16750.166,E2 16750.166} C_VEL
LIN {X 0,Y 355.923,Z 653.092,A -85,B 0,C 180,E1 16747.587,E2 16747.587} C_VEL
LIN {X 0,Y 355.229,Z 656.063,A -85,B 0,C 180,E1 16745.005,E2 16745.005} C_VEL
LIN {X 0,Y 354.762,Z 657.308,A -85,B 0,C 180,E1 16742.422,E2 16742.422} C_VEL
LIN {X 0,Y 354.474,Z 656.807,A -85,B 0,C 180,E1 16739.676,E2 16739.676} C_VEL
LIN {X 0,Y 354.369,Z 654.634,A -85,B 0,C 180,E1 16737.088,E2 16737.088} C_VEL
LIN {X 0,Y 354.446,Z 650.727,A -85,B 0,C 180,E1 16734.496,E2 16734.496} C_VEL
LIN {X 0,Y 354.734,Z 645.048,A -85,B 0,C 180,E1 16731.898,E2 16731.898} C_VEL
LIN {X 0,Y 355.238,Z 637.96,A -85,B 0,C 180,E1 16729.458,E2 16729.458} C_VEL
LIN {X 0,Y 355.965,Z 628.841,A -85,B 0,C 180,E1 16727.014,E2 16727.014} C_VEL
LIN {X 0,Y 356.901,Z 618.201,A -85,B 0,C 180,E1 16724.731,E2 16724.731} C_VEL
LIN {X 0,Y 358.013,Z 606.062,A -85,B 0,C 180,E1 16722.612,E2 16722.612} C_VEL
LIN {X 0,Y 359.224,Z 592.215,A -85,B 0,C 180,E1 16720.656,E2 16720.656} C_VEL
LIN {X 0,Y 360.459,Z 577.107,A -85,B 0,C 180,E1 16718.921,E2 16718.921} C_VEL
LIN {X 0,Y 361.588,Z 561.103,A -85,B 0,C 180,E1 16717.455,E2 16717.455} C_VEL
LIN {X 0,Y 362.614,Z 543.195,A -85,B 0,C 180,E1 16716.174,E2 16716.174} C_VEL
LIN {X 0,Y 363.142,Z 531.718,A -85,B 0,C 180,E1 16715.519,E2 16715.519} C_VEL
LIN {X 0,Y 364.423,Z 532.712,A -85,B 0,C 180,E1 16715.178,E2 16715.178} C_VEL
LIN {X 0,Y 366.628,Z 531.69,A -85,B 0,C 180,E1 16714.821,E2 16714.821} C_VEL
LIN {X 0,Y 369.783,Z 528.153,A -85,B 0,C 180,E1 16714.482,E2 16714.482} C_VEL
LIN {X 0,Y 373.096,Z 522.656,A -85,B 0,C 180,E1 16714.269,E2 16714.269} C_VEL
LIN {X 0,Y 376.513,Z 520.373,A -85,B 0,C 180,E1 16713.799,E2 16713.799} C_VEL
LIN {X 0,Y 380.135,Z 516.029,A -85,B 0,C 180,E1 16713.439,E2 16713.439} C_VEL
LIN {X 0,Y 384.205,Z 508.287,A -85,B 0,C 180,E1 16713.187,E2 16713.187} C_VEL
LIN {X 0,Y 385.939,Z 504.164,A -85,B 0,C 180,E1 16713.122,E2 16713.122} C_VEL
LIN {X 0,Y 389.845,Z 499.585,A -85,B 0,C 180,E1 16712.692,E2 16712.692} C_VEL
LIN {X 0,Y 393.828,Z 492.293,A -85,B 0,C 180,E1 16712.366,E2 16712.366} C_VEL
LIN {X 0,Y 397.849,Z 482.011,A -85,B 0,C 180,E1 16712.136,E2 16712.136} C_VEL
LIN {X 0,Y 396.105,Z 506.086,A -85,B 0,C 180,E1 16711.385,E2 16711.385} C_VEL
LIN {X 0,Y 393.926,Z 526.235,A -85,B 0,C 180,E1 16710.5,E2 16710.5} C_VEL
LIN {X 0,Y 391.224,Z 545.227,A -85,B 0,C 180,E1 16709.43,E2 16709.43} C_VEL
LIN {X 0,Y 387.762,Z 564.869,A -85,B 0,C 180,E1 16708.032,E2 16708.032} C_VEL
LIN {X 0,Y 383.945,Z 583.068,A -85,B 0,C 180,E1 16706.443,E2 16706.443} C_VEL
LIN {X 0,Y 379.719,Z 600.983,A -85,B 0,C 180,E1 16704.548,E2 16704.548} C_VEL
LIN {X 0,Y 375.216,Z 618.496,A -85,B 0,C 180,E1 16702.32,E2 16702.32} C_VEL
LIN {X 0,Y 370.944,Z 634.031,A -85,B 0,C 180,E1 16699.953,E2 16699.953} C_VEL
LIN {X 0,Y 366.733,Z 648.916,A -85,B 0,C 180,E1 16697.244,E2 16697.244} C_VEL
LIN {X 0,Y 362.799,Z 662.701,A -85,B 0,C 180,E1 16694.229,E2 16694.229} C_VEL
LIN {X 0,Y 359.447,Z 674.753,A -85,B 0,C 180,E1 16691.032,E2 16691.032} C_VEL
LIN {X 0,Y 356.852,Z 684.808,A -85,B 0,C 180,E1 16687.801,E2 16687.801} C_VEL
LIN {X 0,Y 354.82,Z 693.661,A -85,B 0,C 180,E1 16684.305,E2 16684.305} C_VEL
LIN {X 0,Y 353.495,Z 700.706,A -85,B 0,C 180,E1 16680.795,E2 16680.795} C_VEL
LIN {X 0,Y 352.794,Z 705.402,A -85,B 0,C 180,E1 16677.757,E2 16677.757} C_VEL
LIN {X 0,Y 351.625,Z 707.104,A -85,B 0,C 180,E1 16676.541,E2 16676.541} C_VEL
LIN {X 0,Y 344.982,Z 710.982,A -85,B 0,C 180,E1 16673.173,E2 16673.173} C_VEL
LIN {X 0,Y 344.285,Z 711.657,A -85,B 0,C 180,E1 16672.165,E2 16672.165} C_VEL
LIN {X 0,Y 344.184,Z 713.062,A -85,B 0,C 180,E1 16668.636,E2 16668.636} C_VEL
LIN {X 0,Y 344.184,Z 713.018,A -85,B 0,C 180,E1 16665.318,E2 16665.318} C_VEL
LIN {X 0,Y 344.261,Z 711.516,A -85,B 0,C 180,E1 16661.824,E2 16661.824} C_VEL
LIN {X 0,Y 344.497,Z 708.626,A -85,B 0,C 180,E1 16658.344,E2 16658.344} C_VEL
LIN {X 0,Y 345.064,Z 704.129,A -85,B 0,C 180,E1 16654.821,E2 16654.821} C_VEL
LIN {X 0,Y 346.07,Z 698.03,A -85,B 0,C 180,E1 16651.325,E2 16651.325} C_VEL
LIN {X 0,Y 347.761,Z 689.877,A -85,B 0,C 180,E1 16647.693,E2 16647.693} C_VEL
LIN {X 0,Y 349.975,Z 680.777,A -85,B 0,C 180,E1 16644.426,E2 16644.426} C_VEL
LIN {X 0,Y 352.868,Z 669.83,A -85,B 0,C 180,E1 16641.199,E2 16641.199} C_VEL
LIN {X 0,Y 356.283,Z 657.382,A -85,B 0,C 180,E1 16638.179,E2 16638.179} C_VEL
LIN {X 0,Y 360.118,Z 643.551,A -85,B 0,C 180,E1 16635.365,E2 16635.365} C_VEL
LIN {X 0,Y 364.311,Z 628.26,A -85,B 0,C 180,E1 16632.758,E2 16632.758} C_VEL
LIN {X 0,Y 368.434,Z 612.494,A -85,B 0,C 180,E1 16630.501,E2 16630.501} C_VEL
LIN {X 0,Y 372.651,Z 595.258,A -85,B 0,C 180,E1 16628.433,E2 16628.433} C_VEL
LIN {X 0,Y 376.644,Z 576.968,A -85,B 0,C 180,E1 16626.618,E2 16626.618} C_VEL
LIN {X 0,Y 380.162,Z 558.666,A -85,B 0,C 180,E1 16625.114,E2 16625.114} C_VEL
LIN {X 0,Y 383.394,Z 538.764,A -85,B 0,C 180,E1 16623.784,E2 16623.784} C_VEL
LIN {X 0,Y 386.068,Z 518.535,A -85,B 0,C 180,E1 16622.716,E2 16622.716} C_VEL
LIN {X 0,Y 388.102,Z 497.476,A -85,B 0,C 180,E1 16621.882,E2 16621.882} C_VEL
LIN {X 0,Y 390.033,Z 467.44,A -85,B 0,C 180,E1 16621.057,E2 16621.057} C_VEL
LIN {X 0,Y 398.504,Z 345.864,A -85,B 0,C 180,E1 16618.236,E2 16618.236} C_VEL
LIN {X 0,Y 402.515,Z 277.635,A -85,B 0,C 180,E1 16616.773,E2 16616.773} C_VEL
LIN {X 0,Y 389.359,Z 261.386,A -85,B 0,C 180,E1 16614.116,E2 16614.116} C_VEL
LIN {X 0,Y 376.498,Z 246.433,A -85,B 0,C 180,E1 16611.271,E2 16611.271} C_VEL
LIN {X 0,Y 369.117,Z 238.376,A -85,B 0,C 180,E1 16609.45,E2 16609.45} C_VEL
LIN {X 0,Y 367.026,Z 234.514,A -85,B 0,C 180,E1 16608.05,E2 16608.05} C_VEL
LIN {X 0,Y 364.928,Z 230.546,A -85,B 0,C 180,E1 16606.551,E2 16606.551} C_VEL
LIN {X 0,Y 362.194,Z 225.668,A -85,B 0,C 180,E1 16604.523,E2 16604.523} C_VEL
LIN {X 0,Y 359.887,Z 221.632,A -85,B 0,C 180,E1 16602.68,E2 16602.68} C_VEL
LIN {X 0,Y 356.877,Z 216.691,A -85,B 0,C 180,E1 16600.106,E2 16600.106} C_VEL
LIN {X 0,Y 356.282,Z 215.456,A -85,B 0,C 180,E1 16599.489,E2 16599.489} C_VEL
LIN {X 0,Y 353.654,Z 211.67,A -85,B 0,C 180,E1 16597.028,E2 16597.028} C_VEL
LIN {X 0,Y 352.993,Z 209.993,A -85,B 0,C 180,E1 16596.098,E2 16596.098} C_VEL
LIN {X 0,Y 350.253,Z 206.52,A -85,B 0,C 180,E1 16593.042,E2 16593.042} C_VEL
LIN {X 0,Y 349.511,Z 204.377,A -85,B 0,C 180,E1 16591.569,E2 16591.569} C_VEL
LIN {X 0,Y 345.924,Z 198.616,A -85,B 0,C 180,E1 16583.148,E2 16583.148} C_VEL
LIN {X 0,Y 345.915,Z 198.621,A -85,B 0,C 180,E1 16578.889,E2 16578.889} C_VEL
LIN {X 0,Y 345.918,Z 198.625,A -85,B 0,C 180,E1 16574.565,E2 16574.565} C_VEL
LIN {X 0,Y 349.78,Z 204.731,A -85,B 0,C 180,E1 16565.864,E2 16565.864} C_VEL
LIN {X 0,Y 351.702,Z 208.787,A -85,B 0,C 180,E1 16562.934,E2 16562.934} C_VEL
LIN {X 0,Y 353.381,Z 210.647,A -85,B 0,C 180,E1 16561.298,E2 16561.298} C_VEL
LIN {X 0,Y 355.38,Z 214.567,A -85,B 0,C 180,E1 16559.033,E2 16559.033} C_VEL
LIN {X 0,Y 356.588,Z 215.932,A -85,B 0,C 180,E1 16558.072,E2 16558.072} C_VEL
LIN {X 0,Y 358.828,Z 220.169,A -85,B 0,C 180,E1 16555.988,E2 16555.988} C_VEL
LIN {X 0,Y 359.817,Z 221.613,A -85,B 0,C 180,E1 16555.219,E2 16555.219} C_VEL
LIN {X 0,Y 361.935,Z 225.459,A -85,B 0,C 180,E1 16553.497,E2 16553.497} C_VEL
LIN {X 0,Y 365.792,Z 232.29,A -85,B 0,C 180,E1 16550.72,E2 16550.72} C_VEL
LIN {X 0,Y 368.488,Z 237.262,A -85,B 0,C 180,E1 16548.893,E2 16548.893} C_VEL
LIN {X 0,Y 372.851,Z 245.325,A -85,B 0,C 180,E1 16546.193,E2 16546.193} C_VEL
LIN {X 0,Y 378.957,Z 257.537,A -85,B 0,C 180,E1 16542.654,E2 16542.654} C_VEL
LIN {X 0,Y 385.134,Z 270.871,A -85,B 0,C 180,E1 16539.325,E2 16539.325} C_VEL
LIN {X 0,Y 391.319,Z 285.156,A -85,B 0,C 180,E1 16536.167,E2 16536.167} C_VEL
LIN {X 0,Y 396.331,Z 297.396,A -85,B 0,C 180,E1 16533.721,E2 16533.721} C_VEL
LIN {X 0,Y 390.212,Z 338.452,A -85,B 0,C 180,E1 16529.713,E2 16529.713} C_VEL
LIN {X 0,Y 389.212,Z 360.003,A -85,B 0,C 180,E1 16527.353,E2 16527.353} C_VEL
LIN {X 0,Y 390.354,Z 379.119,A -85,B 0,C 180,E1 16525.05,E2 16525.05} C_VEL
LIN {X 0,Y 393.69,Z 397.589,A -85,B 0,C 180,E1 16522.628,E2 16522.628} C_VEL
LIN {X 0,Y 399.02,Z 414.204,A -85,B 0,C 180,E1 16520.285,E2 16520.285} C_VEL
LIN {X 0,Y 406.819,Z 430.275,A -85,B 0,C 180,E1 16517.859,E2 16517.859} C_VEL
LIN {X 0,Y 407.193,Z 431.464,A -85,B 0,C 180,E1 16517.706,E2 16517.706} C_VEL
LIN {X 0,Y 402.518,Z 440.162,A -85,B 0,C 180,E1 16517.369,E2 16517.369} C_VEL
LIN {X 0,Y 397.636,Z 468.071,A -85,B 0,C 180,E1 16517.355,E2 16517.355} C_VEL
LIN {X 0,Y 394.653,Z 490.089,A -85,B 0,C 180,E1 16517.116,E2 16517.116} C_VEL
LIN {X 0,Y 392.298,Z 511.564,A -85,B 0,C 180,E1 16516.571,E2 16516.571} C_VEL
LIN {X 0,Y 388.712,Z 538.046,A -85,B 0,C 180,E1 16515.663,E2 16515.663} C_VEL
LIN {X 0,Y 384.448,Z 563.985,A -85,B 0,C 180,E1 16514.5,E2 16514.5} C_VEL
LIN {X 0,Y 380.159,Z 587.705,A -85,B 0,C 180,E1 16513.143,E2 16513.143} C_VEL
LIN {X 0,Y 375.686,Z 610.709,A -85,B 0,C 180,E1 16511.506,E2 16511.506} C_VEL
LIN {X 0,Y 371.26,Z 632.038,A -85,B 0,C 180,E1 16509.663,E2 16509.663} C_VEL
LIN {X 0,Y 367.111,Z 651.172,A -85,B 0,C 180,E1 16507.694,E2 16507.694} C_VEL
LIN {X 0,Y 363.093,Z 668.888,A -85,B 0,C 180,E1 16505.523,E2 16505.523} C_VEL
LIN {X 0,Y 358.759,Z 687.195,A -85,B 0,C 180,E1 16502.824,E2 16502.824} C_VEL
LIN {X 0,Y 355.265,Z 701.978,A -85,B 0,C 180,E1 16500.23,E2 16500.23} C_VEL
LIN {X 0,Y 351.938,Z 716.462,A -85,B 0,C 180,E1 16497.219,E2 16497.219} C_VEL
LIN {X 0,Y 349.276,Z 728.728,A -85,B 0,C 180,E1 16494.164,E2 16494.164} C_VEL
LIN {X 0,Y 347.084,Z 740.169,A -85,B 0,C 180,E1 16490.752,E2 16490.752} C_VEL
LIN {X 0,Y 345.53,Z 749.851,A -85,B 0,C 180,E1 16487.167,E2 16487.167} C_VEL
LIN {X 0,Y 344.652,Z 757.165,A -85,B 0,C 180,E1 16483.762,E2 16483.762} C_VEL
LIN {X 0,Y 344.221,Z 762.968,A -85,B 0,C 180,E1 16480.206,E2 16480.206} C_VEL
LIN {X 0,Y 344.123,Z 766.843,A -85,B 0,C 180,E1 16476.841,E2 16476.841} C_VEL
LIN {X 0,Y 344.144,Z 769.121,A -85,B 0,C 180,E1 16473.498,E2 16473.498} C_VEL
LIN {X 0,Y 344.175,Z 769.912,A -85,B 0,C 180,E1 16470.166,E2 16470.166} C_VEL
LIN {X 0,Y 344.157,Z 769.188,A -85,B 0,C 180,E1 16466.835,E2 16466.835} C_VEL
LIN {X 0,Y 344.126,Z 766.945,A -85,B 0,C 180,E1 16463.493,E2 16463.493} C_VEL
LIN {X 0,Y 344.209,Z 763.178,A -85,B 0,C 180,E1 16460.131,E2 16460.131} C_VEL
LIN {X 0,Y 344.569,Z 757.775,A -85,B 0,C 180,E1 16456.747,E2 16456.747} C_VEL
LIN {X 0,Y 345.408,Z 750.304,A -85,B 0,C 180,E1 16453.173,E2 16453.173} C_VEL
LIN {X 0,Y 346.8,Z 741.29,A -85,B 0,C 180,E1 16449.759,E2 16449.759} C_VEL
LIN {X 0,Y 348.877,Z 730.305,A -85,B 0,C 180,E1 16446.344,E2 16446.344} C_VEL
LIN {X 0,Y 351.588,Z 717.733,A -85,B 0,C 180,E1 16443.117,E2 16443.117} C_VEL
LIN {X 0,Y 354.883,Z 703.706,A -85,B 0,C 180,E1 16440.087,E2 16440.087} C_VEL
LIN {X 0,Y 358.681,Z 688.11,A -85,B 0,C 180,E1 16437.262,E2 16437.262} C_VEL
LIN {X 0,Y 362.941,Z 670.87,A -85,B 0,C 180,E1 16434.631,E2 16434.631} C_VEL
LIN {X 0,Y 367.288,Z 652.792,A -85,B 0,C 180,E1 16432.327,E2 16432.327} C_VEL
LIN {X 0,Y 371.847,Z 632.896,A -85,B 0,C 180,E1 16430.211,E2 16430.211} C_VEL
LIN {X 0,Y 376.739,Z 610.134,A -85,B 0,C 180,E1 16428.229,E2 16428.229} C_VEL
LIN {X 0,Y 381.553,Z 586.615,A -85,B 0,C 180,E1 16426.541,E2 16426.541} C_VEL
LIN {X 0,Y 385.999,Z 563.685,A -85,B 0,C 180,E1 16425.205,E2 16425.205} C_VEL
LIN {X 0,Y 390.632,Z 537.537,A -85,B 0,C 180,E1 16424.007,E2 16424.007} C_VEL
LIN {X 0,Y 394.908,Z 508.755,A -85,B 0,C 180,E1 16422.996,E2 16422.996} C_VEL
LIN {X 0,Y 397.514,Z 487.996,A -85,B 0,C 180,E1 16422.452,E2 16422.452} C_VEL
LIN {X 0,Y 400.467,Z 464.808,A -85,B 0,C 180,E1 16422.118,E2 16422.118} C_VEL
LIN {X 0,Y 404.166,Z 433.901,A -85,B 0,C 180,E1 16421.911,E2 16421.911} C_VEL
LIN {X 0,Y 405.984,Z 422.758,A -85,B 0,C 180,E1 16421.893,E2 16421.893} C_VEL
LIN {X 0,Y 416.747,Z 393.53,A -85,B 0,C 180,E1 16421.014,E2 16421.014} C_VEL
LIN {X 0,Y 427.814,Z 367.703,A -85,B 0,C 180,E1 16420.47,E2 16420.47} C_VEL
LIN {X 0,Y 432.362,Z 357.603,A -85,B 0,C 180,E1 16420.293,E2 16420.293} C_VEL
LIN {X 0,Y 424.773,Z 345.235,A -85,B 0,C 180,E1 16418.247,E2 16418.247} C_VEL
LIN {X 0,Y 420.945,Z 337.133,A -85,B 0,C 180,E1 16416.98,E2 16416.98} C_VEL
LIN {X 0,Y 406.638,Z 346.674,A -85,B 0,C 180,E1 16415.47,E2 16415.47} C_VEL
LIN {X 0,Y 400.511,Z 350.958,A -85,B 0,C 180,E1 16414.781,E2 16414.781} C_VEL
LIN {X 0,Y 394.982,Z 354.846,A -85,B 0,C 180,E1 16414.129,E2 16414.129} C_VEL
LIN {X 0,Y 389.677,Z 358.612,A -85,B 0,C 180,E1 16413.481,E2 16413.481} C_VEL
LIN {X 0,Y 382.956,Z 364.284,A -85,B 0,C 180,E1 16412.714,E2 16412.714} C_VEL
LIN {X 0,Y 375.324,Z 374.542,A -85,B 0,C 180,E1 16412.194,E2 16412.194} C_VEL
LIN {X 0,Y 372.863,Z 377.135,A -85,B 0,C 180,E1 16411.899,E2 16411.899} C_VEL
LIN {X 0,Y 364.84,Z 468.765,A -85,B 0,C 180,E1 16408.972,E2 16408.972} C_VEL
LIN {X 0,Y 362.209,Z 513.012,A -85,B 0,C 180,E1 16407.579,E2 16407.579} C_VEL
LIN {X 0,Y 361.582,Z 536.994,A -85,B 0,C 180,E1 16406.693,E2 16406.693} C_VEL
LIN {X 0,Y 360.891,Z 554.247,A -85,B 0,C 180,E1 16405.783,E2 16405.783} C_VEL
LIN {X 0,Y 359.756,Z 571.47,A -85,B 0,C 180,E1 16404.55,E2 16404.55} C_VEL
LIN {X 0,Y 358.466,Z 586.714,A -85,B 0,C 180,E1 16403.159,E2 16403.159} C_VEL
LIN {X 0,Y 356.86,Z 601.457,A -85,B 0,C 180,E1 16401.446,E2 16401.446} C_VEL
LIN {X 0,Y 355.28,Z 613.914,A -85,B 0,C 180,E1 16399.651,E2 16399.651} C_VEL
LIN {X 0,Y 353.598,Z 625.224,A -85,B 0,C 180,E1 16397.611,E2 16397.611} C_VEL
LIN {X 0,Y 352.046,Z 634.686,A -85,B 0,C 180,E1 16395.484,E2 16395.484} C_VEL
LIN {X 0,Y 350.62,Z 642.758,A -85,B 0,C 180,E1 16393.187,E2 16393.187} C_VEL
LIN {X 0,Y 349.356,Z 649.298,A -85,B 0,C 180,E1 16390.721,E2 16390.721} C_VEL
LIN {X 0,Y 348.278,Z 654.266,A -85,B 0,C 180,E1 16388.086,E2 16388.086} C_VEL
LIN {X 0,Y 347.501,Z 657.407,A -85,B 0,C 180,E1 16385.448,E2 16385.448} C_VEL
LIN {X 0,Y 346.96,Z 658.747,A -85,B 0,C 180,E1 16382.807,E2 16382.807} C_VEL
LIN {X 0,Y 346.631,Z 658.398,A -85,B 0,C 180,E1 16380.165,E2 16380.165} C_VEL
LIN {X 0,Y 346.476,Z 656.235,A -85,B 0,C 180,E1 16377.353,E2 16377.353} C_VEL
LIN {X 0,Y 346.533,Z 652.434,A -85,B 0,C 180,E1 16374.702,E2 16374.702} C_VEL
LIN {X 0,Y 346.804,Z 646.821,A -85,B 0,C 180,E1 16372.045,E2 16372.045} C_VEL
LIN {X 0,Y 347.345,Z 639.279,A -85,B 0,C 180,E1 16369.383,E2 16369.383} C_VEL
LIN {X 0,Y 348.095,Z 630.111,A -85,B 0,C 180,E1 16366.884,E2 16366.884} C_VEL
LIN {X 0,Y 349.065,Z 619.427,A -85,B 0,C 180,E1 16364.55,E2 16364.55} C_VEL
LIN {X 0,Y 350.218,Z 607.237,A -85,B 0,C 180,E1 16362.384,E2 16362.384} C_VEL
LIN {X 0,Y 351.472,Z 593.309,A -85,B 0,C 180,E1 16360.385,E2 16360.385} C_VEL
LIN {X 0,Y 352.735,Z 578.383,A -85,B 0,C 180,E1 16358.638,E2 16358.638} C_VEL
LIN {X 0,Y 353.907,Z 562.355,A -85,B 0,C 180,E1 16357.14,E2 16357.14} C_VEL
LIN {X 0,Y 354.93,Z 545.98,A -85,B 0,C 180,E1 16355.912,E2 16355.912} C_VEL
LIN {X 0,Y 355.964,Z 546.748,A -85,B 0,C 180,E1 16355.612,E2 16355.612} C_VEL
LIN {X 0,Y 358.034,Z 546.141,A -85,B 0,C 180,E1 16355.234,E2 16355.234} C_VEL
LIN {X 0,Y 360.696,Z 543.912,A -85,B 0,C 180,E1 16354.904,E2 16354.904} C_VEL
LIN {X 0,Y 363.903,Z 540.015,A -85,B 0,C 180,E1 16354.619,E2 16354.619} C_VEL
LIN {X 0,Y 367.39,Z 538.175,A -85,B 0,C 180,E1 16354.099,E2 16354.099} C_VEL
LIN {X 0,Y 371.511,Z 534.199,A -85,B 0,C 180,E1 16353.666,E2 16353.666} C_VEL
LIN {X 0,Y 375.742,Z 528.42,A -85,B 0,C 180,E1 16353.359,E2 16353.359} C_VEL
LIN {X 0,Y 380.183,Z 524.54,A -85,B 0,C 180,E1 16352.851,E2 16352.851} C_VEL
LIN {X 0,Y 384.517,Z 518.85,A -85,B 0,C 180,E1 16352.5,E2 16352.5} C_VEL
LIN {X 0,Y 388.94,Z 510.398,A -85,B 0,C 180,E1 16352.281,E2 16352.281} C_VEL
LIN {X 0,Y 389.959,Z 508.449,A -85,B 0,C 180,E1 16352.22,E2 16352.22} C_VEL
LIN {X 0,Y 390.41,Z 508.105,A -85,B 0,C 180,E1 16352.165,E2 16352.165} C_VEL
LIN {X 0,Y 387.949,Z 529.463,A -85,B 0,C 180,E1 16351.198,E2 16351.198} C_VEL
LIN {X 0,Y 384.914,Z 549.235,A -85,B 0,C 180,E1 16350.033,E2 16350.033} C_VEL
LIN {X 0,Y 381.506,Z 567.487,A -85,B 0,C 180,E1 16348.693,E2 16348.693} C_VEL
LIN {X 0,Y 377.326,Z 586.236,A -85,B 0,C 180,E1 16347.002,E2 16347.002} C_VEL
LIN {X 0,Y 373.01,Z 603.562,A -85,B 0,C 180,E1 16345.109,E2 16345.109} C_VEL
LIN {X 0,Y 368.46,Z 620.263,A -85,B 0,C 180,E1 16342.921,E2 16342.921} C_VEL
LIN {X 0,Y 364.004,Z 635.629,A -85,B 0,C 180,E1 16340.522,E2 16340.522} C_VEL
LIN {X 0,Y 359.795,Z 649.745,A -85,B 0,C 180,E1 16337.901,E2 16337.901} C_VEL
LIN {X 0,Y 355.674,Z 663.293,A -85,B 0,C 180,E1 16334.879,E2 16334.879} C_VEL
LIN {X 0,Y 352.178,Z 675.115,A -85,B 0,C 180,E1 16331.696,E2 16331.696} C_VEL
LIN {X 0,Y 349.347,Z 685.349,A -85,B 0,C 180,E1 16328.351,E2 16328.351} C_VEL
LIN {X 0,Y 347.138,Z 694.261,A -85,B 0,C 180,E1 16324.771,E2 16324.771} C_VEL
LIN {X 0,Y 345.744,Z 701.012,A -85,B 0,C 180,E1 16321.369,E2 16321.369} C_VEL
LIN {X 0,Y 344.862,Z 706.352,A -85,B 0,C 180,E1 16317.826,E2 16317.826} C_VEL
LIN {X 0,Y 344.415,Z 710.12,A -85,B 0,C 180,E1 16314.276,E2 16314.276} C_VEL
LIN {X 0,Y 344.285,Z 711.657,A -85,B 0,C 180,E1 16312.165,E2 16312.165} C_VEL
LIN {X 0,Y 343.235,Z 712.452,A -85,B 0,C 180,E1 16310.89,E2 16310.89} C_VEL
LIN {X 0,Y 338.569,Z 713.598,A -85,B 0,C 180,E1 16308.477,E2 16308.477} C_VEL
LIN {X 0,Y 336.345,Z 713.868,A -85,B 0,C 180,E1 16306.806,E2 16306.806} C_VEL
LIN {X 0,Y 336.208,Z 713.81,A -85,B 0,C 180,E1 16306.33,E2 16306.33} C_VEL
LIN {X 0,Y 336.252,Z 712.859,A -85,B 0,C 180,E1 16302.887,E2 16302.887} C_VEL
LIN {X 0,Y 336.436,Z 710.375,A -85,B 0,C 180,E1 16299.359,E2 16299.359} C_VEL
LIN {X 0,Y 336.94,Z 706.207,A -85,B 0,C 180,E1 16295.62,E2 16295.62} C_VEL
LIN {X 0,Y 337.88,Z 700.639,A -85,B 0,C 180,E1 16292.035,E2 16292.035} C_VEL
LIN {X 0,Y 339.406,Z 693.369,A -85,B 0,C 180,E1 16288.481,E2 16288.481} C_VEL
LIN {X 0,Y 341.495,Z 684.779,A -85,B 0,C 180,E1 16285.129,E2 16285.129} C_VEL
LIN {X 0,Y 344.449,Z 673.877,A -85,B 0,C 180,E1 16281.655,E2 16281.655} C_VEL
LIN {X 0,Y 347.811,Z 662.129,A -85,B 0,C 180,E1 16278.559,E2 16278.559} C_VEL
LIN {X 0,Y 351.669,Z 649.045,A -85,B 0,C 180,E1 16275.679,E2 16275.679} C_VEL
LIN {X 0,Y 356.112,Z 633.57,A -85,B 0,C 180,E1 16272.854,E2 16272.854} C_VEL
LIN {X 0,Y 360.412,Z 617.904,A -85,B 0,C 180,E1 16270.471,E2 16270.471} C_VEL
LIN {X 0,Y 364.826,Z 600.782,A -85,B 0,C 180,E1 16268.285,E2 16268.285} C_VEL
LIN {X 0,Y 369.093,Z 582.633,A -85,B 0,C 180,E1 16266.364,E2 16266.364} C_VEL
LIN {X 0,Y 372.896,Z 564.433,A -85,B 0,C 180,E1 16264.765,E2 16264.765} C_VEL
LIN {X 0,Y 376.438,Z 544.312,A -85,B 0,C 180,E1 16263.328,E2 16263.328} C_VEL
LIN {X 0,Y 379.314,Z 523.997,A -85,B 0,C 180,E1 16262.189,E2 16262.189} C_VEL
LIN {X 0,Y 381.53,Z 503.3,A -85,B 0,C 180,E1 16261.299,E2 16261.299} C_VEL
LIN {X 0,Y 383.398,Z 477.68,A -85,B 0,C 180,E1 16260.523,E2 16260.523} C_VEL
LIN {X 0,Y 392.213,Z 357,A -85,B 0,C 180,E1 16257.643,E2 16257.643} C_VEL
LIN {X 0,Y 396.849,Z 281.731,A -85,B 0,C 180,E1 16255.988,E2 16255.988} C_VEL
LIN {X 0,Y 385.11,Z 267.109,A -85,B 0,C 180,E1 16253.535,E2 16253.535} C_VEL
LIN {X 0,Y 372.73,Z 252.644,A -85,B 0,C 180,E1 16250.723,E2 16250.723} C_VEL
LIN {X 0,Y 363.083,Z 241.932,A -85,B 0,C 180,E1 16248.27,E2 16248.27} C_VEL
LIN {X 0,Y 360.135,Z 236.701,A -85,B 0,C 180,E1 16246.208,E2 16246.208} C_VEL
LIN {X 0,Y 357.442,Z 231.868,A -85,B 0,C 180,E1 16244.149,E2 16244.149} C_VEL
LIN {X 0,Y 354.764,Z 227.091,A -85,B 0,C 180,E1 16241.91,E2 16241.91} C_VEL
LIN {X 0,Y 352.494,Z 223.237,A -85,B 0,C 180,E1 16239.871,E2 16239.871} C_VEL
LIN {X 0,Y 351.724,Z 221.925,A -85,B 0,C 180,E1 16239.131,E2 16239.131} C_VEL
LIN {X 0,Y 349.352,Z 218.178,A -85,B 0,C 180,E1 16236.739,E2 16236.739} C_VEL
LIN {X 0,Y 348.844,Z 216.818,A -85,B 0,C 180,E1 16235.986,E2 16235.986} C_VEL
LIN {X 0,Y 346.083,Z 213.17,A -85,B 0,C 180,E1 16232.784,E2 16232.784} C_VEL
LIN {X 0,Y 345.357,Z 211.196,A -85,B 0,C 180,E1 16231.343,E2 16231.343} C_VEL
LIN {X 0,Y 341.943,Z 205.554,A -85,B 0,C 180,E1 16223.069,E2 16223.069} C_VEL
LIN {X 0,Y 341.435,Z 205.263,A -85,B 0,C 180,E1 16217.029,E2 16217.029} C_VEL
LIN {X 0,Y 341.997,Z 205.845,A -85,B 0,C 180,E1 16214.217,E2 16214.217} C_VEL
LIN {X 0,Y 345.698,Z 211.643,A -85,B 0,C 180,E1 16205.977,E2 16205.977} C_VEL
LIN {X 0,Y 347.661,Z 215.7,A -85,B 0,C 180,E1 16202.968,E2 16202.968} C_VEL
LIN {X 0,Y 349.153,Z 217.389,A -85,B 0,C 180,E1 16201.477,E2 16201.477} C_VEL
LIN {X 0,Y 351.13,Z 221.284,A -85,B 0,C 180,E1 16199.185,E2 16199.185} C_VEL
LIN {X 0,Y 352.277,Z 222.732,A -85,B 0,C 180,E1 16198.211,E2 16198.211} C_VEL
LIN {X 0,Y 354.742,Z 227.112,A -85,B 0,C 180,E1 16195.96,E2 16195.96} C_VEL
LIN {X 0,Y 358.211,Z 233.314,A -85,B 0,C 180,E1 16193.107,E2 16193.107} C_VEL
LIN {X 0,Y 361.177,Z 238.725,A -85,B 0,C 180,E1 16190.922,E2 16190.922} C_VEL
LIN {X 0,Y 365.537,Z 246.659,A -85,B 0,C 180,E1 16188.002,E2 16188.002} C_VEL
LIN {X 0,Y 371.096,Z 257.857,A -85,B 0,C 180,E1 16184.53,E2 16184.53} C_VEL
LIN {X 0,Y 376.786,Z 269.751,A -85,B 0,C 180,E1 16181.272,E2 16181.272} C_VEL
LIN {X 0,Y 382.864,Z 283.612,A -85,B 0,C 180,E1 16177.985,E2 16177.985} C_VEL
LIN {X 0,Y 389.489,Z 299.598,A -85,B 0,C 180,E1 16174.615,E2 16174.615} C_VEL
LIN {X 0,Y 390.114,Z 301.595,A -85,B 0,C 180,E1 16174.252,E2 16174.252} C_VEL
LIN {X 0,Y 384.052,Z 340.534,A -85,B 0,C 180,E1 16170.406,E2 16170.406} C_VEL
LIN {X 0,Y 382.826,Z 362.401,A -85,B 0,C 180,E1 16167.982,E2 16167.982} C_VEL
LIN {X 0,Y 383.809,Z 382.096,A -85,B 0,C 180,E1 16165.577,E2 16165.577} C_VEL
LIN {X 0,Y 387.025,Z 400.866,A -85,B 0,C 180,E1 16163.084,E2 16163.084} C_VEL
LIN {X 0,Y 392.393,Z 418.114,A -85,B 0,C 180,E1 16160.619,E2 16160.619} C_VEL
LIN {X 0,Y 399.346,Z 433.367,A -85,B 0,C 180,E1 16158.309,E2 16158.309} C_VEL
LIN {X 0,Y 397.314,Z 437.326,A -85,B 0,C 180,E1 16158.167,E2 16158.167} C_VEL
LIN {X 0,Y 392.823,Z 462.155,A -85,B 0,C 180,E1 16158.186,E2 16158.186} C_VEL
LIN {X 0,Y 389.864,Z 482.374,A -85,B 0,C 180,E1 16158.031,E2 16158.031} C_VEL
LIN {X 0,Y 387.453,Z 501.258,A -85,B 0,C 180,E1 16157.66,E2 16157.66} C_VEL
LIN {X 0,Y 383.837,Z 530.01,A -85,B 0,C 180,E1 16156.731,E2 16156.731} C_VEL
LIN {X 0,Y 379.689,Z 555.23,A -85,B 0,C 180,E1 16155.685,E2 16155.685} C_VEL
LIN {X 0,Y 375.272,Z 579.406,A -85,B 0,C 180,E1 16154.378,E2 16154.378} C_VEL
LIN {X 0,Y 370.601,Z 603.01,A -85,B 0,C 180,E1 16152.791,E2 16152.791} C_VEL
LIN {X 0,Y 365.956,Z 625.186,A -85,B 0,C 180,E1 16150.974,E2 16150.974} C_VEL
LIN {X 0,Y 361.536,Z 645.24,A -85,B 0,C 180,E1 16149.002,E2 16149.002} C_VEL
LIN {X 0,Y 356.865,Z 664.999,A -85,B 0,C 180,E1 16146.639,E2 16146.639} C_VEL
LIN {X 0,Y 352.768,Z 681.784,A -85,B 0,C 180,E1 16144.236,E2 16144.236} C_VEL
LIN {X 0,Y 348.713,Z 698.105,A -85,B 0,C 180,E1 16141.456,E2 16141.456} C_VEL
LIN {X 0,Y 345.218,Z 712.377,A -85,B 0,C 180,E1 16138.548,E2 16138.548} C_VEL
LIN {X 0,Y 342.09,Z 725.937,A -85,B 0,C 180,E1 16135.26,E2 16135.26} C_VEL
LIN {X 0,Y 339.627,Z 737.715,A -85,B 0,C 180,E1 16131.774,E2 16131.774} C_VEL
LIN {X 0,Y 337.98,Z 746.949,A -85,B 0,C 180,E1 16128.454,E2 16128.454} C_VEL
LIN {X 0,Y 336.857,Z 755.084,A -85,B 0,C 180,E1 16124.789,E2 16124.789} C_VEL
LIN {X 0,Y 336.32,Z 761.052,A -85,B 0,C 180,E1 16121.315,E2 16121.315} C_VEL
LIN {X 0,Y 336.143,Z 765.495,A -85,B 0,C 180,E1 16117.692,E2 16117.692} C_VEL
LIN {X 0,Y 336.156,Z 768.143,A -85,B 0,C 180,E1 16114.264,E2 16114.264} C_VEL
LIN {X 0,Y 336.198,Z 769.205,A -85,B 0,C 180,E1 16110.852,E2 16110.852} C_VEL
LIN {X 0,Y 336.187,Z 768.788,A -85,B 0,C 180,E1 16107.443,E2 16107.443} C_VEL
LIN {X 0,Y 336.146,Z 766.884,A -85,B 0,C 180,E1 16104.024,E2 16104.024} C_VEL
LIN {X 0,Y 336.2,Z 763.393,A -85,B 0,C 180,E1 16100.586,E2 16100.586} C_VEL
LIN {X 0,Y 336.537,Z 758.046,A -85,B 0,C 180,E1 16096.95,E2 16096.95} C_VEL
LIN {X 0,Y 337.305,Z 751.216,A -85,B 0,C 180,E1 16093.467,E2 16093.467} C_VEL
LIN {X 0,Y 338.755,Z 742.131,A -85,B 0,C 180,E1 16089.797,E2 16089.797} C_VEL
LIN {X 0,Y 340.871,Z 731.434,A -85,B 0,C 180,E1 16086.305,E2 16086.305} C_VEL
LIN {X 0,Y 343.784,Z 718.709,A -85,B 0,C 180,E1 16082.868,E2 16082.868} C_VEL
LIN {X 0,Y 347.238,Z 704.758,A -85,B 0,C 180,E1 16079.741,E2 16079.741} C_VEL
LIN {X 0,Y 351.275,Z 689.202,A -85,B 0,C 180,E1 16076.806,E2 16076.806} C_VEL
LIN {X 0,Y 355.716,Z 672.156,A -85,B 0,C 180,E1 16074.122,E2 16074.122} C_VEL
LIN {X 0,Y 360.315,Z 654.196,A -85,B 0,C 180,E1 16071.749,E2 16071.749} C_VEL
LIN {X 0,Y 364.822,Z 635.586,A -85,B 0,C 180,E1 16069.699,E2 16069.699} C_VEL
LIN {X 0,Y 370.269,Z 611.549,A -85,B 0,C 180,E1 16067.538,E2 16067.538} C_VEL
LIN {X 0,Y 375.249,Z 588.388,A -85,B 0,C 180,E1 16065.831,E2 16065.831} C_VEL
LIN {X 0,Y 380.079,Z 564.383,A -85,B 0,C 180,E1 16064.407,E2 16064.407} C_VEL
LIN {X 0,Y 384.836,Z 538.888,A -85,B 0,C 180,E1 16063.208,E2 16063.208} C_VEL
LIN {X 0,Y 389.27,Z 511.105,A -85,B 0,C 180,E1 16062.194,E2 16062.194} C_VEL
LIN {X 0,Y 392.141,Z 489.203,A -85,B 0,C 180,E1 16061.593,E2 16061.593} C_VEL
LIN {X 0,Y 395.406,Z 465.139,A -85,B 0,C 180,E1 16061.221,E2 16061.221} C_VEL
LIN {X 0,Y 399.225,Z 433.644,A -85,B 0,C 180,E1 16061.014,E2 16061.014} C_VEL
LIN {X 0,Y 401.482,Z 419.497,A -85,B 0,C 180,E1 16061.009,E2 16061.009} C_VEL
LIN {X 0,Y 410.675,Z 394.412,A -85,B 0,C 180,E1 16060.246,E2 16060.246} C_VEL
LIN {X 0,Y 421.697,Z 368.521,A -85,B 0,C 180,E1 16059.699,E2 16059.699} C_VEL
LIN {X 0,Y 425.242,Z 360.595,A -85,B 0,C 180,E1 16059.561,E2 16059.561} C_VEL
LIN {X 0,Y 418.378,Z 348.427,A -85,B 0,C 180,E1 16057.546,E2 16057.546} C_VEL
LIN {X 0,Y 417.284,Z 346.233,A -85,B 0,C 180,E1 16057.187,E2 16057.187} C_VEL
LIN {X 0,Y 395.487,Z 361.176,A -85,B 0,C 180,E1 16054.845,E2 16054.845} C_VEL
LIN {X 0,Y 388.51,Z 366.324,A -85,B 0,C 180,E1 16054.035,E2 16054.035} C_VEL
LIN {X 0,Y 384.684,Z 369.569,A -85,B 0,C 180,E1 16053.615,E2 16053.615} C_VEL
LIN {X 0,Y 377.057,Z 379.523,A -85,B 0,C 180,E1 16053.11,E2 16053.11} C_VEL
LIN {X 0,Y 375.126,Z 381.708,A -85,B 0,C 180,E1 16052.938,E2 16052.938} C_VEL
LIN {X 0,Y 370.578,Z 388.988,A -85,B 0,C 180,E1 16052.758,E2 16052.758} C_VEL
LIN {X 0,Y 368.901,Z 391.686,A -85,B 0,C 180,E1 16052.617,E2 16052.617} C_VEL
LIN {X 0,Y 364.979,Z 405.401,A -85,B 0,C 180,E1 16051.942,E2 16051.942} C_VEL
LIN {X 0,Y 357.174,Z 491.517,A -85,B 0,C 180,E1 16049.103,E2 16049.103} C_VEL
LIN {X 0,Y 355.378,Z 530.237,A -85,B 0,C 180,E1 16047.762,E2 16047.762} C_VEL
LIN {X 0,Y 354.665,Z 549.346,A -85,B 0,C 180,E1 16046.857,E2 16046.857} C_VEL
LIN {X 0,Y 353.577,Z 566.488,A -85,B 0,C 180,E1 16045.726,E2 16045.726} C_VEL
LIN {X 0,Y 352.259,Z 582.253,A -85,B 0,C 180,E1 16044.392,E2 16044.392} C_VEL
LIN {X 0,Y 350.509,Z 598.263,A -85,B 0,C 180,E1 16042.649,E2 16042.649} C_VEL
LIN {X 0,Y 348.918,Z 610.509,A -85,B 0,C 180,E1 16040.989,E2 16040.989} C_VEL
LIN {X 0,Y 347.114,Z 622.379,A -85,B 0,C 180,E1 16038.995,E2 16038.995} C_VEL
LIN {X 0,Y 345.347,Z 632.716,A -85,B 0,C 180,E1 16036.829,E2 16036.829} C_VEL
LIN {X 0,Y 343.7,Z 641.562,A -85,B 0,C 180,E1 16034.488,E2 16034.488} C_VEL
LIN {X 0,Y 342.211,Z 648.774,A -85,B 0,C 180,E1 16031.972,E2 16031.972} C_VEL
LIN {X 0,Y 341.017,Z 654.12,A -85,B 0,C 180,E1 16029.45,E2 16029.45} C_VEL
LIN {X 0,Y 340.037,Z 657.931,A -85,B 0,C 180,E1 16026.754,E2 16026.754} C_VEL
LIN {X 0,Y 339.334,Z 659.9,A -85,B 0,C 180,E1 16024.055,E2 16024.055} C_VEL
LIN {X 0,Y 338.858,Z 660.155,A -85,B 0,C 180,E1 16021.183,E2 16021.183} C_VEL
LIN {X 0,Y 338.627,Z 658.67,A -85,B 0,C 180,E1 16018.477,E2 16018.477} C_VEL
LIN {X 0,Y 338.586,Z 655.46,A -85,B 0,C 180,E1 16015.766,E2 16015.766} C_VEL
LIN {X 0,Y 338.785,Z 650.139,A -85,B 0,C 180,E1 16012.879,E2 16012.879} C_VEL
LIN {X 0,Y 339.244,Z 643.177,A -85,B 0,C 180,E1 16010.157,E2 16010.157} C_VEL
LIN {X 0,Y 339.944,Z 634.479,A -85,B 0,C 180,E1 16007.555,E2 16007.555} C_VEL
LIN {X 0,Y 340.913,Z 623.918,A -85,B 0,C 180,E1 16005.042,E2 16005.042} C_VEL
LIN {X 0,Y 342.069,Z 611.832,A -85,B 0,C 180,E1 16002.741,E2 16002.741} C_VEL
LIN {X 0,Y 343.377,Z 598.098,A -85,B 0,C 180,E1 16000.612,E2 16000.612} C_VEL
LIN {X 0,Y 344.703,Z 583.121,A -85,B 0,C 180,E1 15998.741,E2 15998.741} C_VEL
LIN {X 0,Y 345.967,Z 567.082,A -85,B 0,C 180,E1 15997.125,E2 15997.125} C_VEL
LIN {X 0,Y 346.632,Z 558.355,A -85,B 0,C 180,E1 15996.362,E2 15996.362} C_VEL
LIN {X 0,Y 348.157,Z 559.021,A -85,B 0,C 180,E1 15995.932,E2 15995.932} C_VEL
LIN {X 0,Y 350.384,Z 558.065,A -85,B 0,C 180,E1 15995.548,E2 15995.548} C_VEL
LIN {X 0,Y 354.125,Z 554.703,A -85,B 0,C 180,E1 15995.121,E2 15995.121} C_VEL
LIN {X 0,Y 355.017,Z 554.004,A -85,B 0,C 180,E1 15995.01,E2 15995.01} C_VEL
LIN {X 0,Y 357.986,Z 552.796,A -85,B 0,C 180,E1 15994.524,E2 15994.524} C_VEL
LIN {X 0,Y 362.015,Z 549.646,A -85,B 0,C 180,E1 15994.038,E2 15994.038} C_VEL
LIN {X 0,Y 365.181,Z 546.358,A -85,B 0,C 180,E1 15993.756,E2 15993.756} C_VEL
LIN {X 0,Y 369.906,Z 543.229,A -85,B 0,C 180,E1 15993.166,E2 15993.166} C_VEL
LIN {X 0,Y 374.552,Z 538.543,A -85,B 0,C 180,E1 15992.741,E2 15992.741} C_VEL
LIN {X 0,Y 377.938,Z 534.045,A -85,B 0,C 180,E1 15992.514,E2 15992.514} C_VEL
LIN {X 0,Y 382.41,Z 530.229,A -85,B 0,C 180,E1 15992.051,E2 15992.051} C_VEL
LIN {X 0,Y 379.322,Z 549.62,A -85,B 0,C 180,E1 15990.905,E2 15990.905} C_VEL
LIN {X 0,Y 375.425,Z 569.517,A -85,B 0,C 180,E1 15989.423,E2 15989.423} C_VEL
LIN {X 0,Y 371.192,Z 587.641,A -85,B 0,C 180,E1 15987.759,E2 15987.759} C_VEL
LIN {X 0,Y 366.622,Z 605.08,A -85,B 0,C 180,E1 15985.818,E2 15985.818} C_VEL
LIN {X 0,Y 361.742,Z 622.104,A -85,B 0,C 180,E1 15983.539,E2 15983.539} C_VEL
LIN {X 0,Y 356.859,Z 638.029,A -85,B 0,C 180,E1 15980.975,E2 15980.975} C_VEL
LIN {X 0,Y 352.248,Z 652.561,A -85,B 0,C 180,E1 15978.159,E2 15978.159} C_VEL
LIN {X 0,Y 348.146,Z 665.416,A -85,B 0,C 180,E1 15975.184,E2 15975.184} C_VEL
LIN {X 0,Y 344.462,Z 677.192,A -85,B 0,C 180,E1 15971.884,E2 15971.884} C_VEL
LIN {X 0,Y 341.454,Z 687.43,A -85,B 0,C 180,E1 15968.374,E2 15968.374} C_VEL
LIN {X 0,Y 339.27,Z 695.698,A -85,B 0,C 180,E1 15964.872,E2 15964.872} C_VEL
LIN {X 0,Y 337.694,Z 702.861,A -85,B 0,C 180,E1 15961.01,E2 15961.01} C_VEL
LIN {X 0,Y 336.844,Z 707.908,A -85,B 0,C 180,E1 15957.393,E2 15957.393} C_VEL
LIN {X 0,Y 336.409,Z 711.422,A -85,B 0,C 180,E1 15953.733,E2 15953.733} C_VEL
LIN {X 0,Y 336.246,Z 713.319,A -85,B 0,C 180,E1 15950.178,E2 15950.178} C_VEL
LIN {X 0,Y 336.205,Z 713.846,A -85,B 0,C 180,E1 15946.589,E2 15946.589} C_VEL
LIN {X 0,Y 336.208,Z 713.81,A -85,B 0,C 180,E1 15946.33,E2 15946.33} C_VEL
LIN {X 0,Y 335.233,Z 713.719,A -85,B 0,C 180,E1 15945.016,E2 15945.016} C_VEL
LIN {X 0,Y 330.841,Z 713.257,A -85,B 0,C 180,E1 15942.625,E2 15942.625} C_VEL
LIN {X 0,Y 328.566,Z 712.425,A -85,B 0,C 180,E1 15940.921,E2 15940.921} C_VEL
LIN {X 0,Y 328.393,Z 711.979,A -85,B 0,C 180,E1 15940.342,E2 15940.342} C_VEL
LIN {X 0,Y 328.775,Z 708.604,A -85,B 0,C 180,E1 15936.812,E2 15936.812} C_VEL
LIN {X 0,Y 329.58,Z 703.576,A -85,B 0,C 180,E1 15933.131,E2 15933.131} C_VEL
LIN {X 0,Y 330.949,Z 696.973,A -85,B 0,C 180,E1 15929.481,E2 15929.481} C_VEL
LIN {X 0,Y 333.019,Z 688.665,A -85,B 0,C 180,E1 15925.868,E2 15925.868} C_VEL
LIN {X 0,Y 335.865,Z 678.404,A -85,B 0,C 180,E1 15922.302,E2 15922.302} C_VEL
LIN {X 0,Y 339.158,Z 667.258,A -85,B 0,C 180,E1 15919.125,E2 15919.125} C_VEL
LIN {X 0,Y 343.155,Z 654.115,A -85,B 0,C 180,E1 15916.005,E2 15916.005} C_VEL
LIN {X 0,Y 347.339,Z 640.36,A -85,B 0,C 180,E1 15913.27,E2 15913.27} C_VEL
LIN {X 0,Y 351.789,Z 625.275,A -85,B 0,C 180,E1 15910.75,E2 15910.75} C_VEL
LIN {X 0,Y 356.383,Z 608.596,A -85,B 0,C 180,E1 15908.437,E2 15908.437} C_VEL
LIN {X 0,Y 360.664,Z 591.658,A -85,B 0,C 180,E1 15906.472,E2 15906.472} C_VEL
LIN {X 0,Y 364.861,Z 573.235,A -85,B 0,C 180,E1 15904.691,E2 15904.691} C_VEL
LIN {X 0,Y 368.637,Z 554.183,A -85,B 0,C 180,E1 15903.183,E2 15903.183} C_VEL
LIN {X 0,Y 371.869,Z 534.573,A -85,B 0,C 180,E1 15901.932,E2 15901.932} C_VEL
LIN {X 0,Y 374.445,Z 514.369,A -85,B 0,C 180,E1 15900.934,E2 15900.934} C_VEL
LIN {X 0,Y 376.302,Z 494.021,A -85,B 0,C 180,E1 15900.18,E2 15900.18} C_VEL
LIN {X 0,Y 380.858,Z 434.176,A -85,B 0,C 180,E1 15898.609,E2 15898.609} C_VEL
LIN {X 0,Y 388.437,Z 333.346,A -85,B 0,C 180,E1 15896.249,E2 15896.249} C_VEL
LIN {X 0,Y 391.402,Z 285.914,A -85,B 0,C 180,E1 15895.214,E2 15895.214} C_VEL
LIN {X 0,Y 378.14,Z 269.558,A -85,B 0,C 180,E1 15892.33,E2 15892.33} C_VEL
LIN {X 0,Y 367.367,Z 257.126,A -85,B 0,C 180,E1 15889.769,E2 15889.769} C_VEL
LIN {X 0,Y 359.027,Z 248.036,A -85,B 0,C 180,E1 15887.616,E2 15887.616} C_VEL
LIN {X 0,Y 356.889,Z 245.655,A -85,B 0,C 180,E1 15886.989,E2 15886.989} C_VEL
LIN {X 0,Y 354.773,Z 241.88,A -85,B 0,C 180,E1 15885.432,E2 15885.432} C_VEL
LIN {X 0,Y 352.977,Z 238.395,A -85,B 0,C 180,E1 15883.948,E2 15883.948} C_VEL
LIN {X 0,Y 350.328,Z 233.636,A -85,B 0,C 180,E1 15881.683,E2 15881.683} C_VEL
LIN {X 0,Y 348.106,Z 229.751,A -85,B 0,C 180,E1 15879.617,E2 15879.617} C_VEL
LIN {X 0,Y 346.894,Z 228.019,A -85,B 0,C 180,E1 15878.506,E2 15878.506} C_VEL
LIN {X 0,Y 344.856,Z 223.923,A -85,B 0,C 180,E1 15876.056,E2 15876.056} C_VEL
LIN {X 0,Y 341.936,Z 219.867,A -85,B 0,C 180,E1 15872.551,E2 15872.551} C_VEL
LIN {X 0,Y 341.306,Z 218.082,A -85,B 0,C 180,E1 15871.234,E2 15871.234} C_VEL
LIN {X 0,Y 338.011,Z 212.52,A -85,B 0,C 180,E1 15862.984,E2 15862.984} C_VEL
LIN {X 0,Y 337.551,Z 212.256,A -85,B 0,C 180,E1 15856.911,E2 15856.911} C_VEL
LIN {X 0,Y 338.073,Z 212.863,A -85,B 0,C 180,E1 15854.21,E2 15854.21} C_VEL
LIN {X 0,Y 341.632,Z 218.617,A -85,B 0,C 180,E1 15846.049,E2 15846.049} C_VEL
LIN {X 0,Y 343.784,Z 222.791,A -85,B 0,C 180,E1 15842.835,E2 15842.835} C_VEL
LIN {X 0,Y 344.931,Z 224.128,A -85,B 0,C 180,E1 15841.662,E2 15841.662} C_VEL
LIN {X 0,Y 347.073,Z 228.219,A -85,B 0,C 180,E1 15839.175,E2 15839.175} C_VEL
LIN {X 0,Y 347.973,Z 229.512,A -85,B 0,C 180,E1 15838.354,E2 15838.354} C_VEL
LIN {X 0,Y 350.46,Z 233.832,A -85,B 0,C 180,E1 15836.074,E2 15836.074} C_VEL
LIN {X 0,Y 353.827,Z 240.163,A -85,B 0,C 180,E1 15833.184,E2 15833.184} C_VEL
LIN {X 0,Y 356.772,Z 245.585,A -85,B 0,C 180,E1 15830.971,E2 15830.971} C_VEL
LIN {X 0,Y 360.64,Z 252.684,A -85,B 0,C 180,E1 15828.324,E2 15828.324} C_VEL
LIN {X 0,Y 366.909,Z 265.325,A -85,B 0,C 180,E1 15824.349,E2 15824.349} C_VEL
LIN {X 0,Y 373.008,Z 278.752,A -85,B 0,C 180,E1 15820.75,E2 15820.75} C_VEL
LIN {X 0,Y 379.216,Z 293.273,A -85,B 0,C 180,E1 15817.36,E2 15817.36} C_VEL
LIN {X 0,Y 383.993,Z 305.346,A -85,B 0,C 180,E1 15814.841,E2 15814.841} C_VEL
LIN {X 0,Y 377.84,Z 343.379,A -85,B 0,C 180,E1 15811.036,E2 15811.036} C_VEL
LIN {X 0,Y 376.478,Z 364.782,A -85,B 0,C 180,E1 15808.632,E2 15808.632} C_VEL
LIN {X 0,Y 377.25,Z 384.614,A -85,B 0,C 180,E1 15806.181,E2 15806.181} C_VEL
LIN {X 0,Y 380.381,Z 404.137,A -85,B 0,C 180,E1 15803.555,E2 15803.555} C_VEL
LIN {X 0,Y 385.404,Z 421.049,A -85,B 0,C 180,E1 15801.104,E2 15801.104} C_VEL
LIN {X 0,Y 391.234,Z 434.166,A -85,B 0,C 180,E1 15799.138,E2 15799.138} C_VEL
LIN {X 0,Y 391.942,Z 435.649,A -85,B 0,C 180,E1 15798.994,E2 15798.994} C_VEL
LIN {X 0,Y 387.653,Z 458.983,A -85,B 0,C 180,E1 15799.021,E2 15799.021} C_VEL
LIN {X 0,Y 384.52,Z 479.285,A -85,B 0,C 180,E1 15798.895,E2 15798.895} C_VEL
LIN {X 0,Y 381.765,Z 499.558,A -85,B 0,C 180,E1 15798.515,E2 15798.515} C_VEL
LIN {X 0,Y 378.035,Z 528.427,A -85,B 0,C 180,E1 15797.579,E2 15797.579} C_VEL
LIN {X 0,Y 373.74,Z 553.779,A -85,B 0,C 180,E1 15796.524,E2 15796.524} C_VEL
LIN {X 0,Y 368.912,Z 579.404,A -85,B 0,C 180,E1 15795.132,E2 15795.132} C_VEL
LIN {X 0,Y 363.968,Z 603.581,A -85,B 0,C 180,E1 15793.484,E2 15793.484} C_VEL
LIN {X 0,Y 359.041,Z 626.191,A -85,B 0,C 180,E1 15791.591,E2 15791.591} C_VEL
LIN {X 0,Y 354.49,Z 645.865,A -85,B 0,C 180,E1 15789.601,E2 15789.601} C_VEL
LIN {X 0,Y 349.841,Z 664.889,A -85,B 0,C 180,E1 15787.294,E2 15787.294} C_VEL
LIN {X 0,Y 345.275,Z 682.677,A -85,B 0,C 180,E1 15784.673,E2 15784.673} C_VEL
LIN {X 0,Y 341.328,Z 697.882,A -85,B 0,C 180,E1 15782.019,E2 15782.019} C_VEL
LIN {X 0,Y 337.479,Z 712.905,A -85,B 0,C 180,E1 15778.876,E2 15778.876} C_VEL
LIN {X 0,Y 334.391,Z 725.61,A -85,B 0,C 180,E1 15775.694,E2 15775.694} C_VEL
LIN {X 0,Y 331.804,Z 737.384,A -85,B 0,C 180,E1 15772.128,E2 15772.128} C_VEL
LIN {X 0,Y 330.074,Z 746.563,A -85,B 0,C 180,E1 15768.729,E2 15768.729} C_VEL
LIN {X 0,Y 328.892,Z 754.679,A -85,B 0,C 180,E1 15764.975,E2 15764.975} C_VEL
LIN {X 0,Y 328.338,Z 760.565,A -85,B 0,C 180,E1 15761.416,E2 15761.416} C_VEL
LIN {X 0,Y 328.159,Z 764.973,A -85,B 0,C 180,E1 15757.704,E2 15757.704} C_VEL
LIN {X 0,Y 328.182,Z 767.549,A -85,B 0,C 180,E1 15754.193,E2 15754.193} C_VEL
LIN {X 0,Y 328.223,Z 768.556,A -85,B 0,C 180,E1 15750.698,E2 15750.698} C_VEL
LIN {X 0,Y 328.21,Z 768.08,A -85,B 0,C 180,E1 15747.206,E2 15747.206} C_VEL
LIN {X 0,Y 328.159,Z 766.095,A -85,B 0,C 180,E1 15743.702,E2 15743.702} C_VEL
LIN {X 0,Y 328.223,Z 762.527,A -85,B 0,C 180,E1 15740.177,E2 15740.177} C_VEL
LIN {X 0,Y 328.612,Z 757.107,A -85,B 0,C 180,E1 15736.45,E2 15736.45} C_VEL
LIN {X 0,Y 329.544,Z 749.805,A -85,B 0,C 180,E1 15732.702,E2 15732.702} C_VEL
LIN {X 0,Y 331.225,Z 740.337,A -85,B 0,C 180,E1 15728.869,E2 15728.869} C_VEL
LIN {X 0,Y 333.675,Z 729.047,A -85,B 0,C 180,E1 15725.196,E2 15725.196} C_VEL
LIN {X 0,Y 336.781,Z 716.569,A -85,B 0,C 180,E1 15721.832,E2 15721.832} C_VEL
LIN {X 0,Y 340.514,Z 702.54,A -85,B 0,C 180,E1 15718.686,E2 15718.686} C_VEL
LIN {X 0,Y 345.065,Z 686.075,A -85,B 0,C 180,E1 15715.595,E2 15715.595} C_VEL
LIN {X 0,Y 349.88,Z 668.565,A -85,B 0,C 180,E1 15712.873,E2 15712.873} C_VEL
LIN {X 0,Y 354.889,Z 649.85,A -85,B 0,C 180,E1 15710.451,E2 15710.451} C_VEL
LIN {X 0,Y 359.779,Z 630.435,A -85,B 0,C 180,E1 15708.378,E2 15708.378} C_VEL
LIN {X 0,Y 365.358,Z 606.364,A -85,B 0,C 180,E1 15706.29,E2 15706.29} C_VEL
LIN {X 0,Y 370.675,Z 582.479,A -85,B 0,C 180,E1 15704.592,E2 15704.592} C_VEL
LIN {X 0,Y 375.752,Z 557.779,A -85,B 0,C 180,E1 15703.188,E2 15703.188} C_VEL
LIN {X 0,Y 380.799,Z 531.031,A -85,B 0,C 180,E1 15702.014,E2 15702.014} C_VEL
LIN {X 0,Y 385.319,Z 501.344,A -85,B 0,C 180,E1 15700.993,E2 15700.993} C_VEL
LIN {X 0,Y 388.589,Z 478.586,A -85,B 0,C 180,E1 15700.477,E2 15700.477} C_VEL
